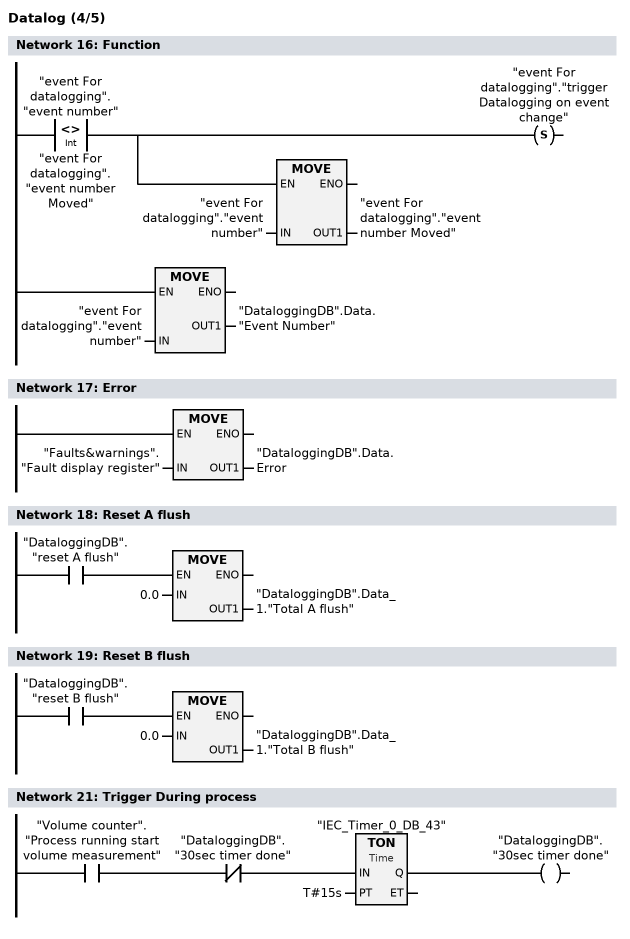
   RUNG wire#powerrail
      { S7_Templates := "SrcType := Int" } NE_Contact(in1 := "event For datalogging"."event number", in2 := "event For datalogging"."event number Moved")
      wire#w1
      S_Coil( "event For datalogging"."trigger Datalogging on event change" )
   END_RUNG
   RUNG wire#w1
      Move(in := "event For datalogging"."event number", out1 => "event For datalogging"."event number Moved")
   END_RUNG
   RUNG wire#powerrail
      Move(in := "event For datalogging"."event number", out1 => "DataloggingDB".Data."Event Number")
   END_RUNG
   // the same network as SCL:
   IF "event For datalogging"."event number" <> "event For datalogging"."event number Moved" THEN
       "event For datalogging"."trigger Datalogging on event change" := TRUE;
       "event For datalogging"."event number Moved" := "event For datalogging"."event number";
   END_IF;
   "DataloggingDB".Data."Event Number" := "event For datalogging"."event number";
END_REGION

REGION Network 17: Error
   RUNG wire#powerrail
      Move(in := "Faults&warnings"."Fault display register", out1 => "DataloggingDB".Data.Error)
   END_RUNG
   // the same network as SCL:
   "DataloggingDB".Data.Error := "Faults&warnings"."Fault display register";
END_REGION

REGION Network 18: Reset A flush
   RUNG wire#powerrail
      Contact( "DataloggingDB"."reset A flush" )
      Move(in := 0.0, out1 => "DataloggingDB".Data_1."Total A flush")
   END_RUNG
   // the same network as SCL:
   IF "DataloggingDB"."reset A flush" THEN "DataloggingDB".Data_1."Total A flush" := 0.0; END_IF;
END_REGION

REGION Network 19: Reset B flush
   RUNG wire#powerrail
      Contact( "DataloggingDB"."reset B flush" )
      Move(in := 0.0, out1 => "DataloggingDB".Data_1."Total B flush")
   END_RUNG
   // the same network as SCL:
   IF "DataloggingDB"."reset B flush" THEN "DataloggingDB".Data_1."Total B flush" := 0.0; END_IF;
END_REGION

REGION Network 20 (SCL): Reset total size
   IF "DataloggingDB"."reset total Size" THEN
       "DataloggingDB".Data_1."Total size A" := 0;
       "DataloggingDB".Data_1."Total size B" := 0;
       "DataloggingDB".totalsizeday := 0;
       "DataloggingDB".totalsizepreviousday := 0;
       "DataloggingDB".totalsizeweek := 0;
       "DataloggingDB".totalsizepreviousweek := 0;
       "DataloggingDB".totalsizemonth := 0;
       "DataloggingDB".totalsizepreviousmonth := 0;
       "DataloggingDB"."reset total Size" := FALSE;
   END_IF;
END_REGION

REGION Network 21: Trigger During process
   RUNG wire#powerrail
      Contact( "Volume counter"."Process running start volume measurement" )
      I_Contact( "DataloggingDB"."30sec timer done" )
      { S7_Templates := "time_type := Time" } "IEC_Timer_0_DB_43".TON(pt := T#15s, et =>)
      Coil( "DataloggingDB"."30sec timer done" )
   END_RUNG
   // the same network as SCL:
   "IEC_Timer_0_DB_43".TON(IN := "Volume counter"."Process running start volume measurement" AND NOT "DataloggingDB"."30sec timer done",
                           PT := T#15s);
   "DataloggingDB"."30sec timer done" := "IEC_Timer_0_DB_43".Q;
END_REGION

REGION Network 22: trigger data logging
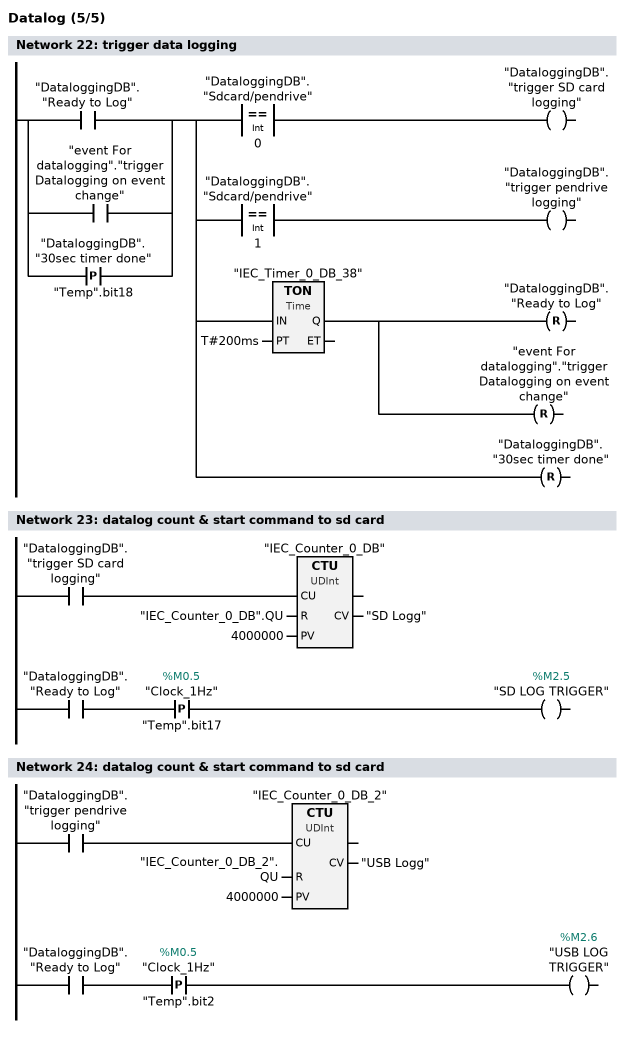
   RUNG wire#powerrail
      Contact( "DataloggingDB"."Ready to Log" )
      wire#w1
      { S7_Templates := "SrcType := Int" } EQ_Contact(in1 := "DataloggingDB"."Sdcard/pendrive", in2 := 0)
      Coil( "DataloggingDB"."trigger SD card logging" )
   END_RUNG
   RUNG wire#powerrail
      Contact( "event For datalogging"."trigger Datalogging on event change" )
   END_RUNG wire#w1
   RUNG wire#powerrail
      P_Contact(operand := "DataloggingDB"."30sec timer done", bit := "Temp".bit18)
   END_RUNG wire#w1
   RUNG wire#w1
      { S7_Templates := "SrcType := Int" } EQ_Contact(in1 := "DataloggingDB"."Sdcard/pendrive", in2 := 1)
      Coil( "DataloggingDB"."trigger pendrive logging" )
   END_RUNG
   RUNG wire#w1
      { S7_Templates := "time_type := Time" } "IEC_Timer_0_DB_38".TON(pt := T#200ms, et =>)
      wire#w2
      R_Coil( "DataloggingDB"."Ready to Log" )
   END_RUNG
   RUNG wire#w2
      R_Coil( "event For datalogging"."trigger Datalogging on event change" )
   END_RUNG
   RUNG wire#w1
      R_Coil( "DataloggingDB"."30sec timer done" )
   END_RUNG
   // the same network as SCL:
   #_w1 := "DataloggingDB"."30sec timer done" AND NOT "Temp".bit18;   // rising edge of "DataloggingDB"."30sec timer done"
   "Temp".bit18 := "DataloggingDB"."30sec timer done";
   #_w2 := "DataloggingDB"."Ready to Log" OR "event For datalogging"."trigger Datalogging on event change" OR #_w1;
   "DataloggingDB"."trigger SD card logging" := #_w2 AND ("DataloggingDB"."Sdcard/pendrive" = 0);
   "DataloggingDB"."trigger pendrive logging" := #_w2 AND ("DataloggingDB"."Sdcard/pendrive" = 1);
   "IEC_Timer_0_DB_38".TON(IN := #_w2, PT := T#200ms);
   IF "IEC_Timer_0_DB_38".Q THEN
       "DataloggingDB"."Ready to Log" := FALSE;
       "event For datalogging"."trigger Datalogging on event change" := FALSE;
   END_IF;
   IF #_w2 THEN "DataloggingDB"."30sec timer done" := FALSE; END_IF;
END_REGION

REGION Network 23: datalog count & start command to sd card
   RUNG wire#powerrail
      Contact( "DataloggingDB"."trigger SD card logging" )
      { S7_Templates := "value_type := UDInt" } "IEC_Counter_0_DB".CTU(r := "IEC_Counter_0_DB".QU, pv := 4000000, cv => "SD Logg")
   END_RUNG
   RUNG wire#powerrail
      Contact( "DataloggingDB"."Ready to Log" )
      P_Contact(operand := "Clock_1Hz", bit := "Temp".bit17)
      Coil( "SD LOG TRIGGER" )
   END_RUNG
   // the same network as SCL:
   "IEC_Counter_0_DB".CTU(CU := "DataloggingDB"."trigger SD card logging",
                          R := "IEC_Counter_0_DB".QU,
                          PV := 4000000,
                          CV => "SD Logg");
   #_w1 := "DataloggingDB"."Ready to Log" AND "Clock_1Hz" AND NOT "Temp".bit17;   // rising edge of "Clock_1Hz"
   "Temp".bit17 := "Clock_1Hz";
   "SD LOG TRIGGER" := #_w1;
END_REGION

REGION Network 24: datalog count & start command to sd card
   RUNG wire#powerrail
      Contact( "DataloggingDB"."trigger pendrive logging" )
      { S7_Templates := "value_type := UDInt" } "IEC_Counter_0_DB_2".CTU(r := "IEC_Counter_0_DB_2".QU, pv := 4000000, cv => "USB Logg")
   END_RUNG
   RUNG wire#powerrail
      Contact( "DataloggingDB"."Ready to Log" )
      P_Contact(operand := "Clock_1Hz", bit := "Temp".bit2)
      Coil( "USB LOG TRIGGER" )
   END_RUNG
   // the same network as SCL:
   "IEC_Counter_0_DB_2".CTU(CU := "DataloggingDB"."trigger pendrive logging",
                           R := "IEC_Counter_0_DB_2".QU,
                           PV := 4000000,
                           CV => "USB Logg");
   #_w1 := "DataloggingDB"."Ready to Log" AND "Clock_1Hz" AND NOT "Temp".bit2;   // rising edge of "Clock_1Hz"
   "Temp".bit2 := "Clock_1Hz";
   "USB LOG TRIGGER" := #_w1;
END_REGION
END_FUNCTION

FUNCTION "IOT_DATA_FC" : Void   // FC1001, LAD
{ S7_Optimized_Access := 'TRUE' }
VERSION : 0.1
// stored: AutoNumber false, IsIECCheckEnabled true, SetENOAutomatically true, UDAEnableTagReadback false
BEGIN

REGION Network 1 (SCL)
   "IOT_DATA"."pump A Inlet" := "pressure"."pump A Inlet";
   "IOT_DATA"."pump B Inlet" := "pressure"."pump B Inlet";
   "IOT_DATA"."pump A Outlet" := "pressure"."pump A Outlet";
   "IOT_DATA"."pump B Outlet" := "pressure"."pump B Outlet";
END_REGION
END_FUNCTION

FUNCTION "Output_Estop" : Void   // FC31, LAD
{ S7_Optimized_Access := 'TRUE' }
VERSION : 0.1
// stored: AutoNumber true, IsIECCheckEnabled false, SetENOAutomatically false, UDAEnableTagReadback false
   VAR_TEMP
      spare : Bool;
      spare2 : Bool;
      spare3 : Bool;
   END_VAR
BEGIN

REGION Network 1: gear Pump A
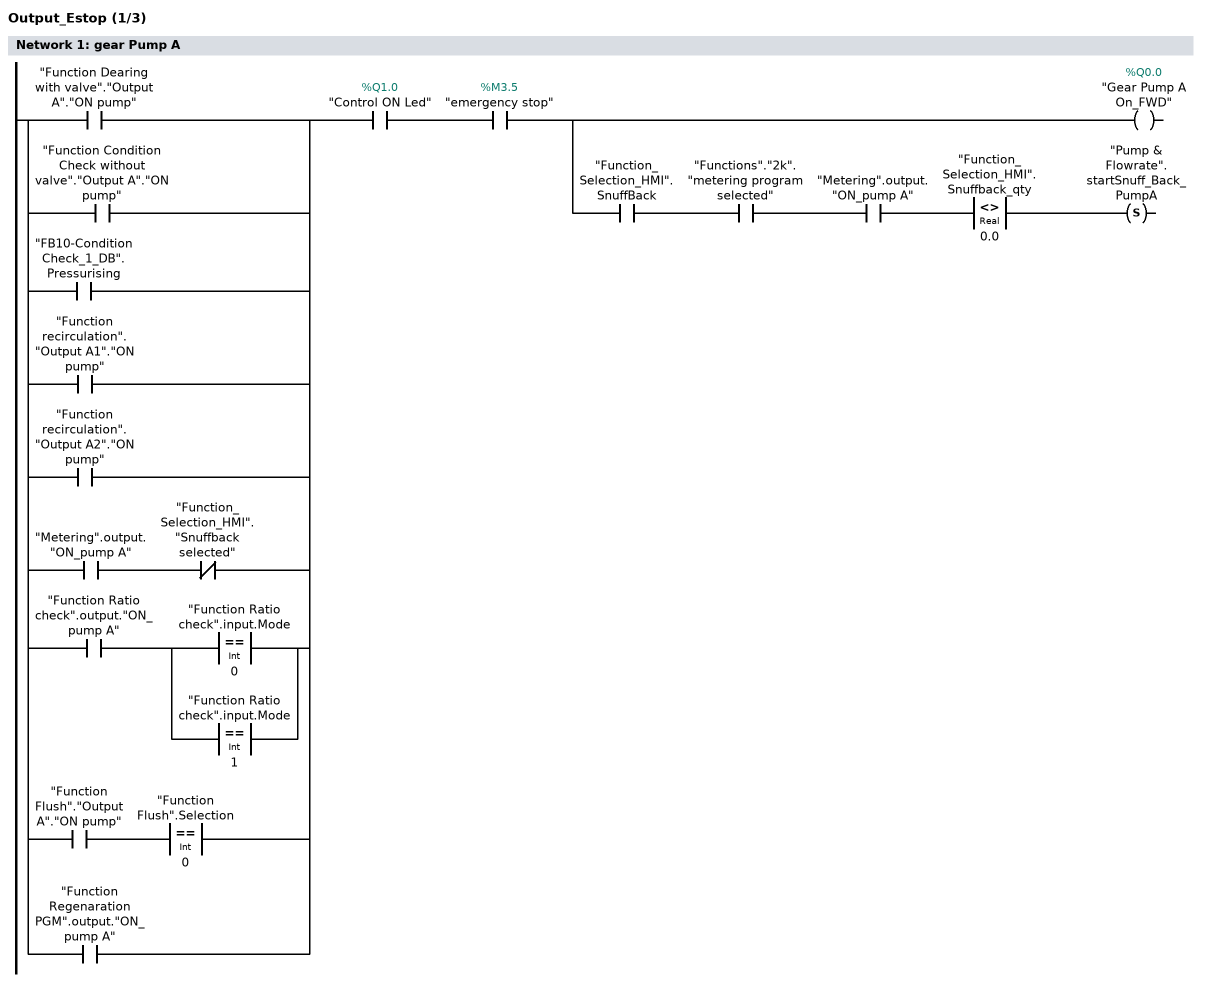
   RUNG wire#powerrail
      Contact( "Function Dearing with valve"."Output A"."ON pump" )
      wire#w1
      Contact( "Control ON Led" )
      Contact( "emergency stop" )
      wire#w3
      Coil( "Gear Pump A On_FWD" )
   END_RUNG
   RUNG wire#powerrail
      Contact( "Function ConditionCheck without valve"."Output A"."ON pump" )
   END_RUNG wire#w1
   RUNG wire#powerrail
      Contact( "FB10-Condition Check_1_DB".Pressurising )
   END_RUNG wire#w1
   RUNG wire#powerrail
      Contact( "Function recirculation"."Output A1"."ON pump" )
   END_RUNG wire#w1
   RUNG wire#powerrail
      Contact( "Function recirculation"."Output A2"."ON pump" )
   END_RUNG wire#w1
   RUNG wire#powerrail
      Contact( "Metering".output."ON_pump A" )
      I_Contact( "Function_Selection_HMI"."Snuffback selected" )
   END_RUNG wire#w1
   RUNG wire#powerrail
      Contact( "Function Ratio check".output."ON_pump A" )
      wire#w2
      { S7_Templates := "SrcType := Int" } EQ_Contact(in1 := "Function Ratio check".input.Mode, in2 := 0)
   END_RUNG wire#w1
   RUNG wire#w2
      { S7_Templates := "SrcType := Int" } EQ_Contact(in1 := "Function Ratio check".input.Mode, in2 := 1)
   END_RUNG wire#w1
   RUNG wire#powerrail
      Contact( "Function Flush"."Output A"."ON pump" )
      { S7_Templates := "SrcType := Int" } EQ_Contact(in1 := "Function Flush".Selection, in2 := 0)
   END_RUNG wire#w1
   RUNG wire#powerrail
      Contact( "Function Regenaration PGM".output."ON_pump A" )
   END_RUNG wire#w1
   RUNG wire#w3
      Contact( "Function_Selection_HMI".SnuffBack )
      Contact( "Functions"."2k"."metering program selected" )
      Contact( "Metering".output."ON_pump A" )
      { S7_Templates := "SrcType := Real" } NE_Contact(in1 := "Function_Selection_HMI".Snuffback_qty, in2 := 0.0)
      S_Coil( "Pump & Flowrate".startSnuff_Back_PumpA )
   END_RUNG
   // the same network as SCL:
   "Gear Pump A On_FWD" := ("Function Dearing with valve"."Output A"."ON pump" OR "Function ConditionCheck without valve"."Output A"."ON pump" OR "FB10-Condition Check_1_DB".Pressurising OR "Function recirculation"."Output A1"."ON pump" OR "Function recirculation"."Output A2"."ON pump" OR ("Metering".output."ON_pump A" AND NOT "Function_Selection_HMI"."Snuffback selected") OR ("Function Ratio check".output."ON_pump A" AND (("Function Ratio check".input.Mode = 0) OR ("Function Ratio check".input.Mode = 1))) OR ("Function Flush"."Output A"."ON pump" AND ("Function Flush".Selection = 0)) OR "Function Regenaration PGM".output."ON_pump A") AND "Control ON Led" AND "emergency stop";
   IF "Gear Pump A On_FWD" AND "Function_Selection_HMI".SnuffBack AND "Functions"."2k"."metering program selected" AND "Metering".output."ON_pump A" AND ("Function_Selection_HMI".Snuffback_qty <> 0.0) THEN
       "Pump & Flowrate".startSnuff_Back_PumpA := TRUE;
   END_IF;
END_REGION

REGION Network 2: gear Pump B
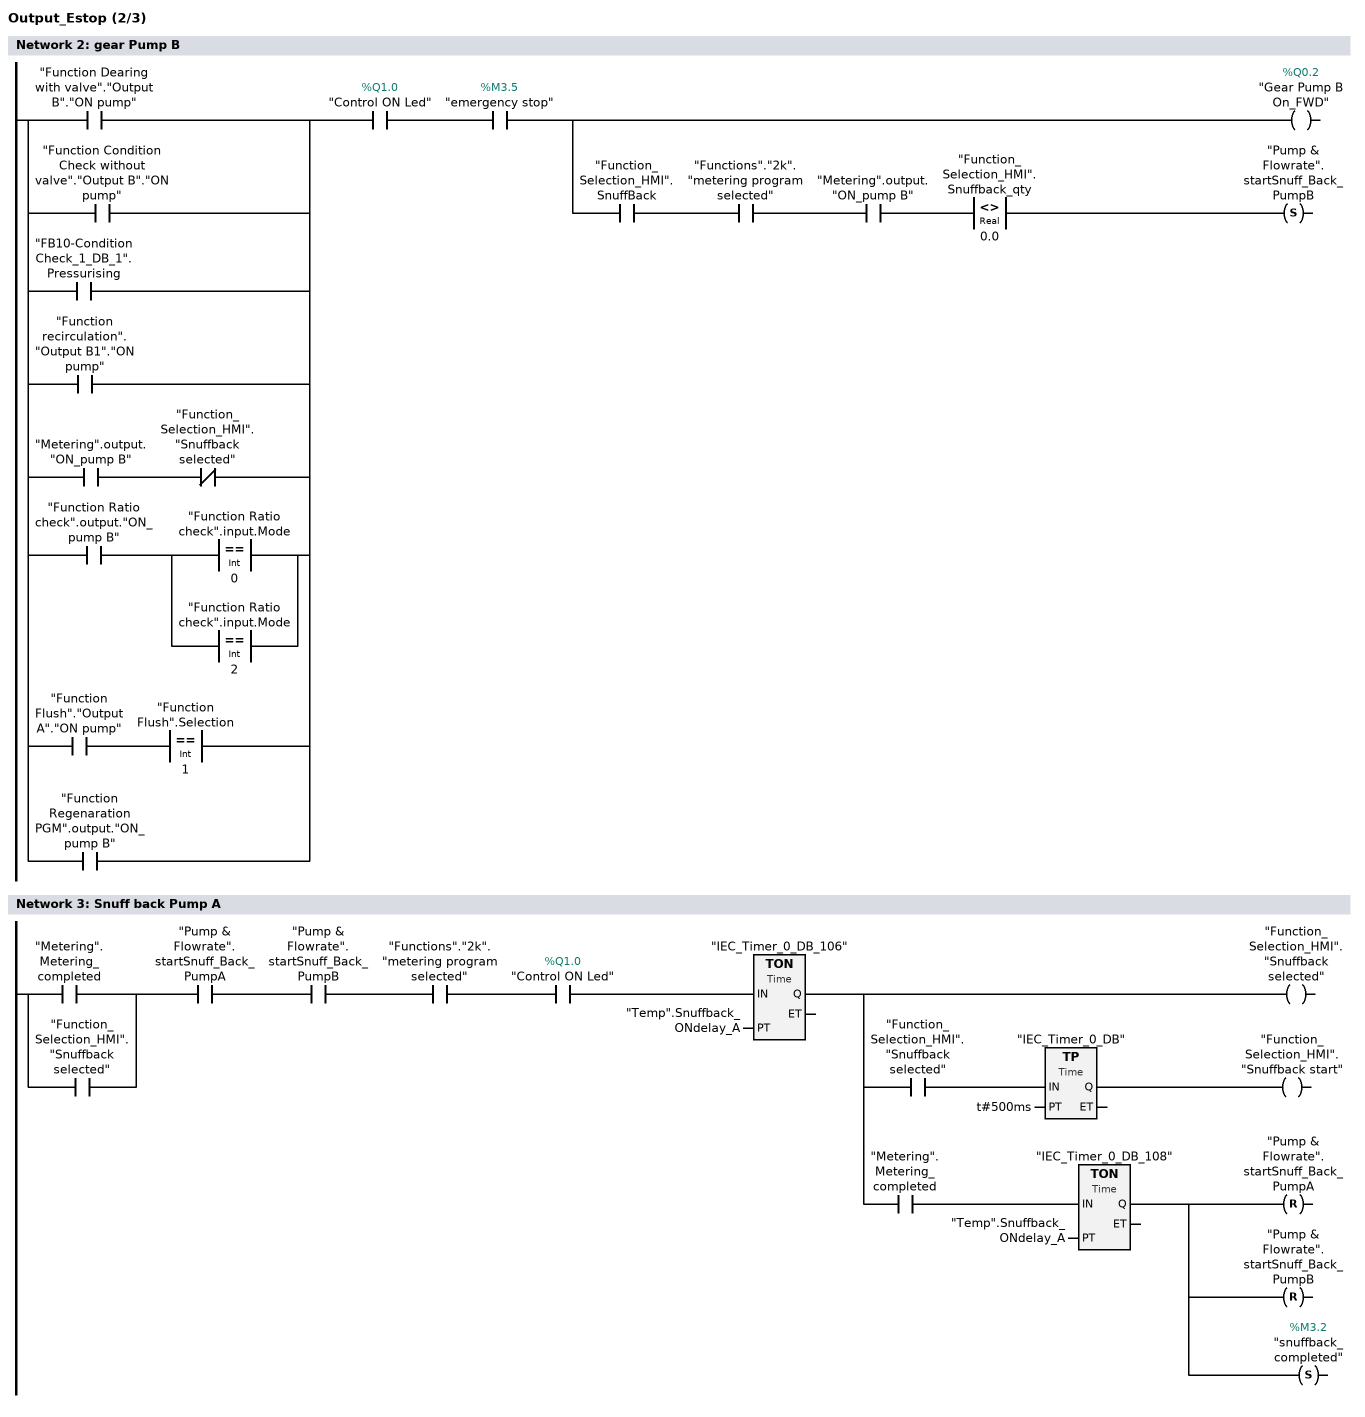
   RUNG wire#powerrail
      Contact( "Function Dearing with valve"."Output B"."ON pump" )
      wire#w1
      Contact( "Control ON Led" )
      Contact( "emergency stop" )
      wire#w3
      Coil( "Gear Pump B On_FWD" )
   END_RUNG
   RUNG wire#powerrail
      Contact( "Function ConditionCheck without valve"."Output B"."ON pump" )
   END_RUNG wire#w1
   RUNG wire#powerrail
      Contact( "FB10-Condition Check_1_DB_1".Pressurising )
   END_RUNG wire#w1
   RUNG wire#powerrail
      Contact( "Function recirculation"."Output B1"."ON pump" )
   END_RUNG wire#w1
   RUNG wire#powerrail
      Contact( "Metering".output."ON_pump B" )
      I_Contact( "Function_Selection_HMI"."Snuffback selected" )
   END_RUNG wire#w1
   RUNG wire#powerrail
      Contact( "Function Ratio check".output."ON_pump B" )
      wire#w2
      { S7_Templates := "SrcType := Int" } EQ_Contact(in1 := "Function Ratio check".input.Mode, in2 := 0)
   END_RUNG wire#w1
   RUNG wire#w2
      { S7_Templates := "SrcType := Int" } EQ_Contact(in1 := "Function Ratio check".input.Mode, in2 := 2)
   END_RUNG wire#w1
   RUNG wire#powerrail
      Contact( "Function Flush"."Output A"."ON pump" )
      { S7_Templates := "SrcType := Int" } EQ_Contact(in1 := "Function Flush".Selection, in2 := 1)
   END_RUNG wire#w1
   RUNG wire#powerrail
      Contact( "Function Regenaration PGM".output."ON_pump B" )
   END_RUNG wire#w1
   RUNG wire#w3
      Contact( "Function_Selection_HMI".SnuffBack )
      Contact( "Functions"."2k"."metering program selected" )
      Contact( "Metering".output."ON_pump B" )
      { S7_Templates := "SrcType := Real" } NE_Contact(in1 := "Function_Selection_HMI".Snuffback_qty, in2 := 0.0)
      S_Coil( "Pump & Flowrate".startSnuff_Back_PumpB )
   END_RUNG
   // the same network as SCL:
   "Gear Pump B On_FWD" := ("Function Dearing with valve"."Output B"."ON pump" OR "Function ConditionCheck without valve"."Output B"."ON pump" OR "FB10-Condition Check_1_DB_1".Pressurising OR "Function recirculation"."Output B1"."ON pump" OR ("Metering".output."ON_pump B" AND NOT "Function_Selection_HMI"."Snuffback selected") OR ("Function Ratio check".output."ON_pump B" AND (("Function Ratio check".input.Mode = 0) OR ("Function Ratio check".input.Mode = 2))) OR ("Function Flush"."Output A"."ON pump" AND ("Function Flush".Selection = 1)) OR "Function Regenaration PGM".output."ON_pump B") AND "Control ON Led" AND "emergency stop";
   IF "Gear Pump B On_FWD" AND "Function_Selection_HMI".SnuffBack AND "Functions"."2k"."metering program selected" AND "Metering".output."ON_pump B" AND ("Function_Selection_HMI".Snuffback_qty <> 0.0) THEN
       "Pump & Flowrate".startSnuff_Back_PumpB := TRUE;
   END_IF;
END_REGION

REGION Network 3: Snuff back Pump A
   RUNG wire#powerrail
      Contact( "Metering".Metering_completed )
      wire#w1
      Contact( "Pump & Flowrate".startSnuff_Back_PumpA )
      Contact( "Pump & Flowrate".startSnuff_Back_PumpB )
      Contact( "Functions"."2k"."metering program selected" )
      Contact( "Control ON Led" )
      { S7_Templates := "time_type := Time" } "IEC_Timer_0_DB_106".TON(pt := "Temp".Snuffback_ONdelay_A, et =>)
      wire#w2
      Coil( "Function_Selection_HMI"."Snuffback selected" )
   END_RUNG
   RUNG wire#powerrail
      Contact( "Function_Selection_HMI"."Snuffback selected" )
   END_RUNG wire#w1
   RUNG wire#w2
      Contact( "Function_Selection_HMI"."Snuffback selected" )
      { S7_Templates := "time_type := Time" } "IEC_Timer_0_DB".TP(pt := t#500ms, et =>)
      Coil( "Function_Selection_HMI"."Snuffback start" )
   END_RUNG
   RUNG wire#w2
      Contact( "Metering".Metering_completed )
      { S7_Templates := "time_type := Time" } "IEC_Timer_0_DB_108".TON(pt := "Temp".Snuffback_ONdelay_A, et =>)
      wire#w3
      R_Coil( "Pump & Flowrate".startSnuff_Back_PumpA )
   END_RUNG
   RUNG wire#w3
      R_Coil( "Pump & Flowrate".startSnuff_Back_PumpB )
   END_RUNG
   RUNG wire#w3
      S_Coil( "snuffback_completed" )
   END_RUNG
   // the same network as SCL:
   "IEC_Timer_0_DB_106".TON(IN := ("Metering".Metering_completed OR "Function_Selection_HMI"."Snuffback selected") AND "Pump & Flowrate".startSnuff_Back_PumpA AND "Pump & Flowrate".startSnuff_Back_PumpB AND "Functions"."2k"."metering program selected" AND "Control ON Led",
                           PT := "Temp".Snuffback_ONdelay_A);
   "Function_Selection_HMI"."Snuffback selected" := "IEC_Timer_0_DB_106".Q;
   "IEC_Timer_0_DB".TP(IN := "IEC_Timer_0_DB_106".Q AND "Function_Selection_HMI"."Snuffback selected",
                       PT := t#500ms);
   "Function_Selection_HMI"."Snuffback start" := "IEC_Timer_0_DB".Q;
   "IEC_Timer_0_DB_108".TON(IN := "IEC_Timer_0_DB_106".Q AND "Metering".Metering_completed,
                           PT := "Temp".Snuffback_ONdelay_A);
   IF "IEC_Timer_0_DB_108".Q THEN
       "Pump & Flowrate".startSnuff_Back_PumpA := FALSE;
       "Pump & Flowrate".startSnuff_Back_PumpB := FALSE;
       "snuffback_completed" := TRUE;
   END_IF;
END_REGION

REGION Network 4
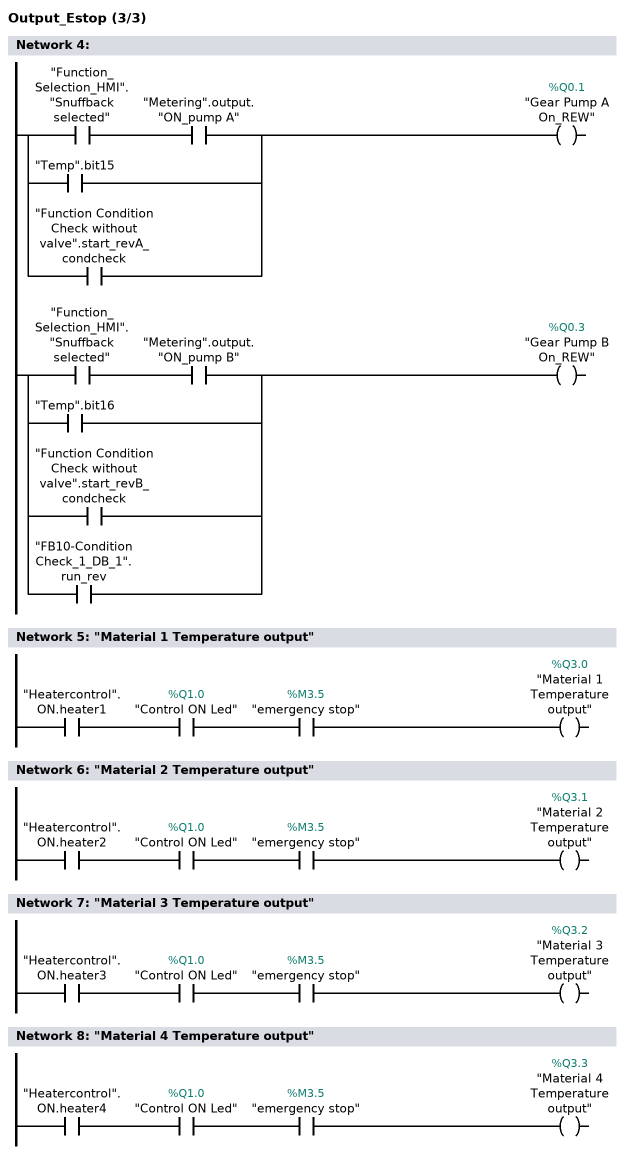
   RUNG wire#powerrail
      Contact( "Function_Selection_HMI"."Snuffback selected" )
      Contact( "Metering".output."ON_pump A" )
      wire#w1
      Coil( "Gear Pump A On_REW" )
   END_RUNG
   RUNG wire#powerrail
      Contact( "Temp".bit15 )
   END_RUNG wire#w1
   RUNG wire#powerrail
      Contact( "Function ConditionCheck without valve".start_revA_condcheck )
   END_RUNG wire#w1
   RUNG wire#powerrail
      Contact( "Function_Selection_HMI"."Snuffback selected" )
      Contact( "Metering".output."ON_pump B" )
      wire#w2
      Coil( "Gear Pump B On_REW" )
   END_RUNG
   RUNG wire#powerrail
      Contact( "Temp".bit16 )
   END_RUNG wire#w2
   RUNG wire#powerrail
      Contact( "Function ConditionCheck without valve".start_revB_condcheck )
   END_RUNG wire#w2
   RUNG wire#powerrail
      Contact( "FB10-Condition Check_1_DB_1".run_rev )
   END_RUNG wire#w2
   // the same network as SCL:
   "Gear Pump A On_REW" := ("Function_Selection_HMI"."Snuffback selected" AND "Metering".output."ON_pump A") OR "Temp".bit15 OR "Function ConditionCheck without valve".start_revA_condcheck;
   "Gear Pump B On_REW" := ("Function_Selection_HMI"."Snuffback selected" AND "Metering".output."ON_pump B") OR "Temp".bit16 OR "Function ConditionCheck without valve".start_revB_condcheck OR "FB10-Condition Check_1_DB_1".run_rev;
END_REGION

REGION Network 5: "Material 1 Temperature output"
   RUNG wire#powerrail
      Contact( "Heatercontrol".ON.heater1 )
      Contact( "Control ON Led" )
      Contact( "emergency stop" )
      Coil( "Material 1 Temperature output" )
   END_RUNG
   // the same network as SCL:
   "Material 1 Temperature output" := "Heatercontrol".ON.heater1 AND "Control ON Led" AND "emergency stop";
END_REGION

REGION Network 6: "Material 2 Temperature output"
   RUNG wire#powerrail
      Contact( "Heatercontrol".ON.heater2 )
      Contact( "Control ON Led" )
      Contact( "emergency stop" )
      Coil( "Material 2 Temperature output" )
   END_RUNG
   // the same network as SCL:
   "Material 2 Temperature output" := "Heatercontrol".ON.heater2 AND "Control ON Led" AND "emergency stop";
END_REGION

REGION Network 7: "Material 3 Temperature output"
   RUNG wire#powerrail
      Contact( "Heatercontrol".ON.heater3 )
      Contact( "Control ON Led" )
      Contact( "emergency stop" )
      Coil( "Material 3 Temperature output" )
   END_RUNG
   // the same network as SCL:
   "Material 3 Temperature output" := "Heatercontrol".ON.heater3 AND "Control ON Led" AND "emergency stop";
END_REGION

REGION Network 8: "Material 4 Temperature output"
   RUNG wire#powerrail
      Contact( "Heatercontrol".ON.heater4 )
      Contact( "Control ON Led" )
      Contact( "emergency stop" )
      Coil( "Material 4 Temperature output" )
   END_RUNG
   // the same network as SCL:
   "Material 4 Temperature output" := "Heatercontrol".ON.heater4 AND "Control ON Led" AND "emergency stop";
END_REGION
END_FUNCTION

FUNCTION "Conditon Check" : Void   // FC11, LAD
{ S7_Optimized_Access := 'TRUE' }
VERSION : 0.1
// stored: AutoNumber true, IsIECCheckEnabled false, SetENOAutomatically false, UDAEnableTagReadback false
   VAR_TEMP   // added for the SCL form of the ladder/FBD networks
      _w1 : Bool;
      _w2 : Bool;
      _w3 : Bool;
   END_VAR
BEGIN

REGION Network 1: Condition Check A without Valve
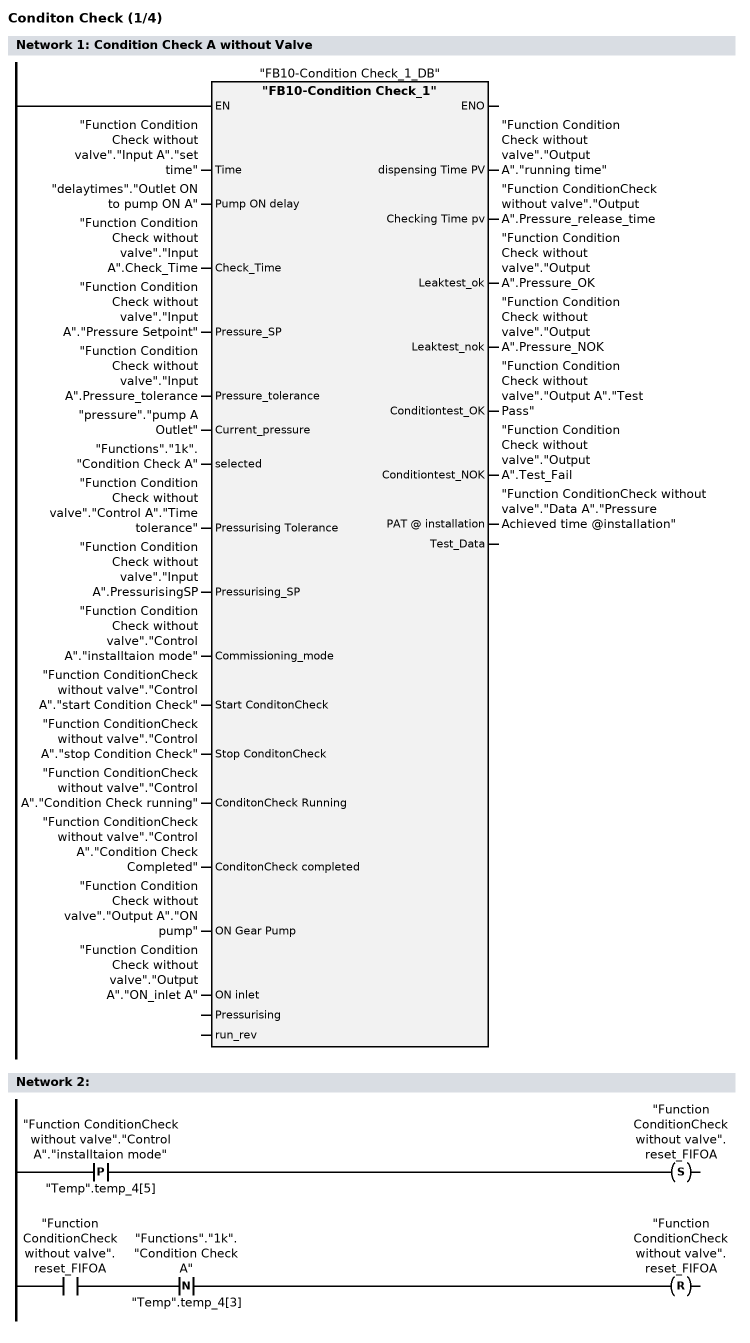
   RUNG wire#powerrail
      "FB10-Condition Check_1_DB"("Time" := "Function ConditionCheck without valve"."Input A"."set time", "Pump ON delay" := "delaytimes"."Outlet ON to pump ON A", Check_Time := "Function ConditionCheck without valve"."Input A".Check_Time, Pressure_SP := "Function ConditionCheck without valve"."Input A"."Pressure Setpoint", Pressure_tolerance := "Function ConditionCheck without valve"."Input A".Pressure_tolerance, Current_pressure := "pressure"."pump A Outlet", selected := "Functions"."1k"."Condition Check A", "Pressurising Tolerance" := "Function ConditionCheck without valve"."Control A"."Time tolerance", Pressurising_SP := "Function ConditionCheck without valve"."Input A".PressurisingSP, Commissioning_mode := "Function ConditionCheck without valve"."Control A"."installtaion mode", "Start ConditonCheck" := "Function ConditionCheck without valve"."Control A"."start Condition Check", "Stop ConditonCheck" := "Function ConditionCheck without valve"."Control A"."stop Condition Check", "ConditonCheck Running" := "Function ConditionCheck without valve"."Control A"."Condition Check running", "ConditonCheck completed" := "Function ConditionCheck without valve"."Control A"."Condition Check Completed", "ON Gear Pump" := "Function ConditionCheck without valve"."Output A"."ON pump", "ON inlet" := "Function ConditionCheck without valve"."Output A"."ON_inlet A", Pressurising :=, run_rev :=, "dispensing Time PV" => "Function ConditionCheck without valve"."Output A"."running time", "Checking Time pv" => "Function ConditionCheck without valve"."Output A".Pressure_release_time, Leaktest_ok => "Function ConditionCheck without valve"."Output A".Pressure_OK, Leaktest_nok => "Function ConditionCheck without valve"."Output A".Pressure_NOK, Conditiontest_OK => "Function ConditionCheck without valve"."Output A"."Test Pass", Conditiontest_NOK => "Function ConditionCheck without valve"."Output A".Test_Fail, "PAT @ installation" => "Function ConditionCheck without valve"."Data A"."Pressure Achieved time @installation", Test_Data =>)
   END_RUNG
   // the same network as SCL:
   "FB10-Condition Check_1_DB"("Time" := "Function ConditionCheck without valve"."Input A"."set time",   // "FB10-Condition Check_1"
                           "Pump ON delay" := "delaytimes"."Outlet ON to pump ON A",
                           Check_Time := "Function ConditionCheck without valve"."Input A".Check_Time,
                           Pressure_SP := "Function ConditionCheck without valve"."Input A"."Pressure Setpoint",
                           Pressure_tolerance := "Function ConditionCheck without valve"."Input A".Pressure_tolerance,
                           Current_pressure := "pressure"."pump A Outlet",
                           selected := "Functions"."1k"."Condition Check A",
                           "Pressurising Tolerance" := "Function ConditionCheck without valve"."Control A"."Time tolerance",
                           Pressurising_SP := "Function ConditionCheck without valve"."Input A".PressurisingSP,
                           Commissioning_mode := "Function ConditionCheck without valve"."Control A"."installtaion mode",
                           "Start ConditonCheck" := "Function ConditionCheck without valve"."Control A"."start Condition Check",
                           "Stop ConditonCheck" := "Function ConditionCheck without valve"."Control A"."stop Condition Check",
                           "ConditonCheck Running" := "Function ConditionCheck without valve"."Control A"."Condition Check running",
                           "ConditonCheck completed" := "Function ConditionCheck without valve"."Control A"."Condition Check Completed",
                           "ON Gear Pump" := "Function ConditionCheck without valve"."Output A"."ON pump",
                           "ON inlet" := "Function ConditionCheck without valve"."Output A"."ON_inlet A",
                           "dispensing Time PV" => "Function ConditionCheck without valve"."Output A"."running time",
                           "Checking Time pv" => "Function ConditionCheck without valve"."Output A".Pressure_release_time,
                           Leaktest_ok => "Function ConditionCheck without valve"."Output A".Pressure_OK,
                           Leaktest_nok => "Function ConditionCheck without valve"."Output A".Pressure_NOK,
                           Conditiontest_OK => "Function ConditionCheck without valve"."Output A"."Test Pass",
                           Conditiontest_NOK => "Function ConditionCheck without valve"."Output A".Test_Fail,
                           "PAT @ installation" => "Function ConditionCheck without valve"."Data A"."Pressure Achieved time @installation");
END_REGION

REGION Network 2
   RUNG wire#powerrail
      P_Contact(operand := "Function ConditionCheck without valve"."Control A"."installtaion mode", bit := "Temp".temp_4[5])
      S_Coil( "Function ConditionCheck without valve".reset_FIFOA )
   END_RUNG
   RUNG wire#powerrail
      Contact( "Function ConditionCheck without valve".reset_FIFOA )
      N_Contact(operand := "Functions"."1k"."Condition Check A", bit := "Temp".temp_4[3])
      R_Coil( "Function ConditionCheck without valve".reset_FIFOA )
   END_RUNG
   // the same network as SCL:
   #_w1 := "Function ConditionCheck without valve"."Control A"."installtaion mode" AND NOT "Temp".temp_4[5];   // rising edge of "Function ConditionCheck without valve"."Control A"."installtaion mode"
   "Temp".temp_4[5] := "Function ConditionCheck without valve"."Control A"."installtaion mode";
   IF #_w1 THEN "Function ConditionCheck without valve".reset_FIFOA := TRUE; END_IF;
   #_w2 := "Function ConditionCheck without valve".reset_FIFOA AND NOT "Functions"."1k"."Condition Check A" AND "Temp".temp_4[3];   // falling edge of "Functions"."1k"."Condition Check A"
   "Temp".temp_4[3] := "Functions"."1k"."Condition Check A";
   IF #_w2 THEN "Function ConditionCheck without valve".reset_FIFOA := FALSE; END_IF;
END_REGION

REGION Network 3
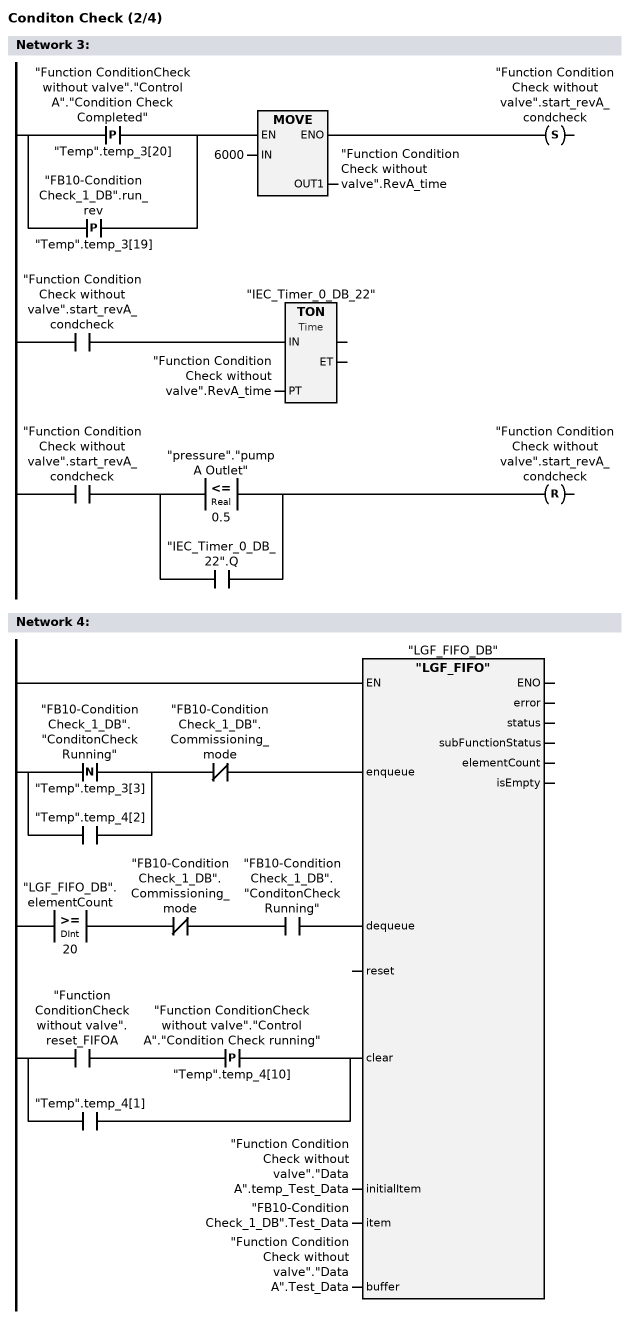
   RUNG wire#powerrail
      P_Contact(operand := "Function ConditionCheck without valve"."Control A"."Condition Check Completed", bit := "Temp".temp_3[20])
      wire#w1
      Move(in := 6000, out1 => "Function ConditionCheck without valve".RevA_time)
      S_Coil( "Function ConditionCheck without valve".start_revA_condcheck )
   END_RUNG
   RUNG wire#powerrail
      P_Contact(operand := "FB10-Condition Check_1_DB".run_rev, bit := "Temp".temp_3[19])
   END_RUNG wire#w1
   RUNG wire#powerrail
      Contact( "Function ConditionCheck without valve".start_revA_condcheck )
      { S7_Templates := "time_type := Time" } "IEC_Timer_0_DB_22".TON(pt := "Function ConditionCheck without valve".RevA_time, et =>)
   END_RUNG
   RUNG wire#powerrail
      Contact( "Function ConditionCheck without valve".start_revA_condcheck )
      wire#w2
      { S7_Templates := "SrcType := Real" } LE_Contact(in1 := "pressure"."pump A Outlet", in2 := 0.5)
      wire#w3
      R_Coil( "Function ConditionCheck without valve".start_revA_condcheck )
   END_RUNG
   RUNG wire#w2
      Contact( "IEC_Timer_0_DB_22".Q )
   END_RUNG wire#w3
   // the same network as SCL:
   #_w1 := "Function ConditionCheck without valve"."Control A"."Condition Check Completed" AND NOT "Temp".temp_3[20];   // rising edge of "Function ConditionCheck without valve"."Control A"."Condition Check Completed"
   "Temp".temp_3[20] := "Function ConditionCheck without valve"."Control A"."Condition Check Completed";
   #_w2 := "FB10-Condition Check_1_DB".run_rev AND NOT "Temp".temp_3[19];   // rising edge of "FB10-Condition Check_1_DB".run_rev
   "Temp".temp_3[19] := "FB10-Condition Check_1_DB".run_rev;
   IF #_w1 OR #_w2 THEN
       "Function ConditionCheck without valve".RevA_time := 6000;
       "Function ConditionCheck without valve".start_revA_condcheck := TRUE;
   END_IF;
   "IEC_Timer_0_DB_22".TON(IN := "Function ConditionCheck without valve".start_revA_condcheck,
                           PT := "Function ConditionCheck without valve".RevA_time);
   IF "Function ConditionCheck without valve".start_revA_condcheck AND (("pressure"."pump A Outlet" <= 0.5) OR "IEC_Timer_0_DB_22".Q) THEN
       "Function ConditionCheck without valve".start_revA_condcheck := FALSE;
   END_IF;
END_REGION

REGION Network 4
   RUNG wire#powerrail
      "LGF_FIFO_DB"(enqueue := wire#w2, dequeue := wire#w3, clear := wire#w4, reset :=, initialItem := "Function ConditionCheck without valve"."Data A".temp_Test_Data, item := "FB10-Condition Check_1_DB".Test_Data, buffer := "Function ConditionCheck without valve"."Data A".Test_Data, error =>, status =>, subFunctionStatus =>, elementCount =>, isEmpty =>)
   END_RUNG
   RUNG wire#powerrail
      N_Contact(operand := "FB10-Condition Check_1_DB"."ConditonCheck Running", bit := "Temp".temp_3[3])
      wire#w1
      I_Contact( "FB10-Condition Check_1_DB".Commissioning_mode )
   END_RUNG wire#w2
   RUNG wire#powerrail
      Contact( "Temp".temp_4[2] )
   END_RUNG wire#w1
   RUNG wire#powerrail
      { S7_Templates := "SrcType := DInt" } GE_Contact(in1 := "LGF_FIFO_DB".elementCount, in2 := 20)
      I_Contact( "FB10-Condition Check_1_DB".Commissioning_mode )
      Contact( "FB10-Condition Check_1_DB"."ConditonCheck Running" )
   END_RUNG wire#w3
   RUNG wire#powerrail
      Contact( "Function ConditionCheck without valve".reset_FIFOA )
      P_Contact(operand := "Function ConditionCheck without valve"."Control A"."Condition Check running", bit := "Temp".temp_4[10])
   END_RUNG wire#w4
   RUNG wire#powerrail
      Contact( "Temp".temp_4[1] )
   END_RUNG wire#w4
   // the same network as SCL:
   #_w1 := NOT "FB10-Condition Check_1_DB"."ConditonCheck Running" AND "Temp".temp_3[3];   // falling edge of "FB10-Condition Check_1_DB"."ConditonCheck Running"
   "Temp".temp_3[3] := "FB10-Condition Check_1_DB"."ConditonCheck Running";
   #_w3 := (#_w1 OR "Temp".temp_4[2]) AND NOT "FB10-Condition Check_1_DB".Commissioning_mode;
   #_w2 := "Function ConditionCheck without valve".reset_FIFOA AND "Function ConditionCheck without valve"."Control A"."Condition Check running" AND NOT "Temp".temp_4[10];   // rising edge of "Function ConditionCheck without valve"."Control A"."Condition Check running"
   "Temp".temp_4[10] := "Function ConditionCheck without valve"."Control A"."Condition Check running";
   "LGF_FIFO_DB"(enqueue := #_w3,   // "LGF_FIFO"
                 dequeue := ("LGF_FIFO_DB".elementCount >= 20) AND NOT "FB10-Condition Check_1_DB".Commissioning_mode AND "FB10-Condition Check_1_DB"."ConditonCheck Running",
                 clear := #_w2 OR "Temp".temp_4[1],
                 initialItem := "Function ConditionCheck without valve"."Data A".temp_Test_Data,
                 item := "FB10-Condition Check_1_DB".Test_Data,
                 buffer := "Function ConditionCheck without valve"."Data A".Test_Data);
END_REGION

REGION Network 5: Condition Check B without Valve
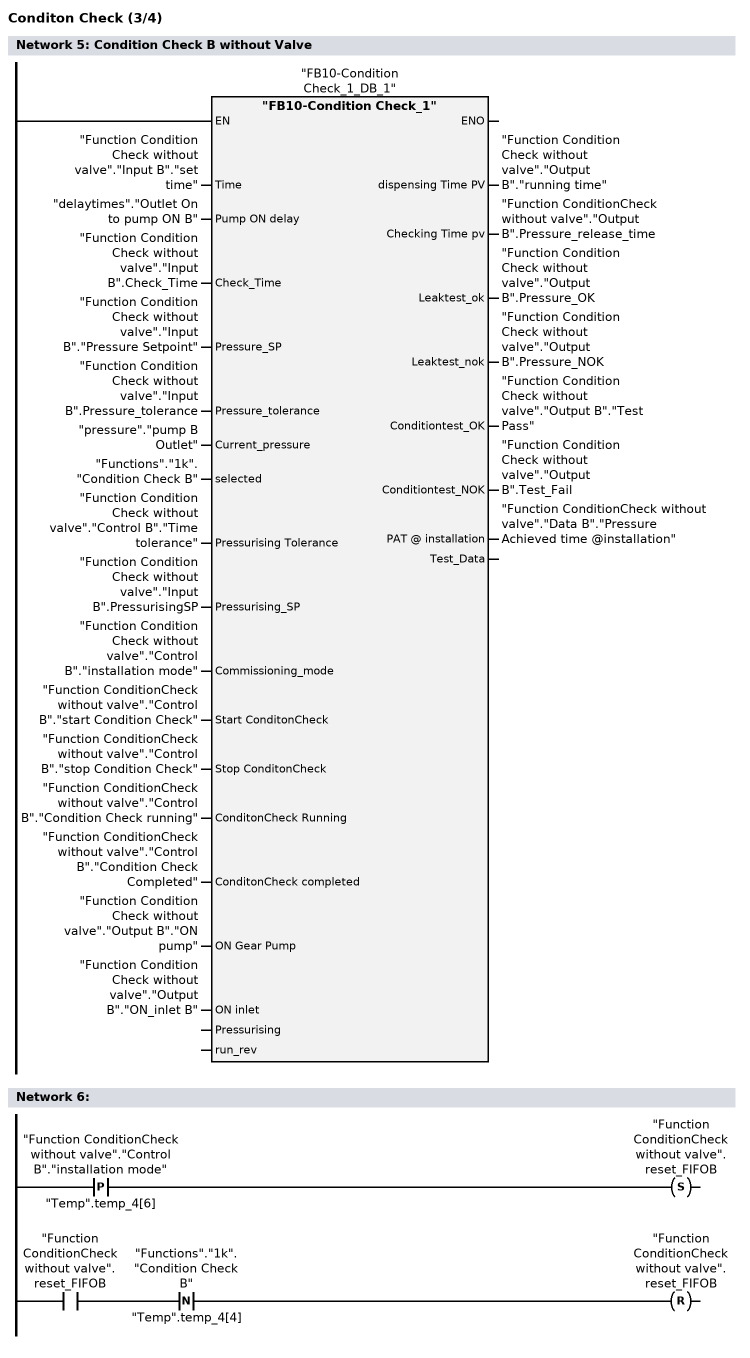
   RUNG wire#powerrail
      "FB10-Condition Check_1_DB_1"("Time" := "Function ConditionCheck without valve"."Input B"."set time", "Pump ON delay" := "delaytimes"."Outlet On to pump ON B", Check_Time := "Function ConditionCheck without valve"."Input B".Check_Time, Pressure_SP := "Function ConditionCheck without valve"."Input B"."Pressure Setpoint", Pressure_tolerance := "Function ConditionCheck without valve"."Input B".Pressure_tolerance, Current_pressure := "pressure"."pump B Outlet", selected := "Functions"."1k"."Condition Check B", "Pressurising Tolerance" := "Function ConditionCheck without valve"."Control B"."Time tolerance", Pressurising_SP := "Function ConditionCheck without valve"."Input B".PressurisingSP, Commissioning_mode := "Function ConditionCheck without valve"."Control B"."installation mode", "Start ConditonCheck" := "Function ConditionCheck without valve"."Control B"."start Condition Check", "Stop ConditonCheck" := "Function ConditionCheck without valve"."Control B"."stop Condition Check", "ConditonCheck Running" := "Function ConditionCheck without valve"."Control B"."Condition Check running", "ConditonCheck completed" := "Function ConditionCheck without valve"."Control B"."Condition Check Completed", "ON Gear Pump" := "Function ConditionCheck without valve"."Output B"."ON pump", "ON inlet" := "Function ConditionCheck without valve"."Output B"."ON_inlet B", Pressurising :=, run_rev :=, "dispensing Time PV" => "Function ConditionCheck without valve"."Output B"."running time", "Checking Time pv" => "Function ConditionCheck without valve"."Output B".Pressure_release_time, Leaktest_ok => "Function ConditionCheck without valve"."Output B".Pressure_OK, Leaktest_nok => "Function ConditionCheck without valve"."Output B".Pressure_NOK, Conditiontest_OK => "Function ConditionCheck without valve"."Output B"."Test Pass", Conditiontest_NOK => "Function ConditionCheck without valve"."Output B".Test_Fail, "PAT @ installation" => "Function ConditionCheck without valve"."Data B"."Pressure Achieved time @installation", Test_Data =>)
   END_RUNG
   // the same network as SCL:
   "FB10-Condition Check_1_DB_1"("Time" := "Function ConditionCheck without valve"."Input B"."set time",   // "FB10-Condition Check_1"
                           "Pump ON delay" := "delaytimes"."Outlet On to pump ON B",
                           Check_Time := "Function ConditionCheck without valve"."Input B".Check_Time,
                           Pressure_SP := "Function ConditionCheck without valve"."Input B"."Pressure Setpoint",
                           Pressure_tolerance := "Function ConditionCheck without valve"."Input B".Pressure_tolerance,
                           Current_pressure := "pressure"."pump B Outlet",
                           selected := "Functions"."1k"."Condition Check B",
                           "Pressurising Tolerance" := "Function ConditionCheck without valve"."Control B"."Time tolerance",
                           Pressurising_SP := "Function ConditionCheck without valve"."Input B".PressurisingSP,
                           Commissioning_mode := "Function ConditionCheck without valve"."Control B"."installation mode",
                           "Start ConditonCheck" := "Function ConditionCheck without valve"."Control B"."start Condition Check",
                           "Stop ConditonCheck" := "Function ConditionCheck without valve"."Control B"."stop Condition Check",
                           "ConditonCheck Running" := "Function ConditionCheck without valve"."Control B"."Condition Check running",
                           "ConditonCheck completed" := "Function ConditionCheck without valve"."Control B"."Condition Check Completed",
                           "ON Gear Pump" := "Function ConditionCheck without valve"."Output B"."ON pump",
                           "ON inlet" := "Function ConditionCheck without valve"."Output B"."ON_inlet B",
                           "dispensing Time PV" => "Function ConditionCheck without valve"."Output B"."running time",
                           "Checking Time pv" => "Function ConditionCheck without valve"."Output B".Pressure_release_time,
                           Leaktest_ok => "Function ConditionCheck without valve"."Output B".Pressure_OK,
                           Leaktest_nok => "Function ConditionCheck without valve"."Output B".Pressure_NOK,
                           Conditiontest_OK => "Function ConditionCheck without valve"."Output B"."Test Pass",
                           Conditiontest_NOK => "Function ConditionCheck without valve"."Output B".Test_Fail,
                           "PAT @ installation" => "Function ConditionCheck without valve"."Data B"."Pressure Achieved time @installation");
END_REGION

REGION Network 6
   RUNG wire#powerrail
      P_Contact(operand := "Function ConditionCheck without valve"."Control B"."installation mode", bit := "Temp".temp_4[6])
      S_Coil( "Function ConditionCheck without valve".reset_FIFOB )
   END_RUNG
   RUNG wire#powerrail
      Contact( "Function ConditionCheck without valve".reset_FIFOB )
      N_Contact(operand := "Functions"."1k"."Condition Check B", bit := "Temp".temp_4[4])
      R_Coil( "Function ConditionCheck without valve".reset_FIFOB )
   END_RUNG
   // the same network as SCL:
   #_w1 := "Function ConditionCheck without valve"."Control B"."installation mode" AND NOT "Temp".temp_4[6];   // rising edge of "Function ConditionCheck without valve"."Control B"."installation mode"
   "Temp".temp_4[6] := "Function ConditionCheck without valve"."Control B"."installation mode";
   IF #_w1 THEN "Function ConditionCheck without valve".reset_FIFOB := TRUE; END_IF;
   #_w2 := "Function ConditionCheck without valve".reset_FIFOB AND NOT "Functions"."1k"."Condition Check B" AND "Temp".temp_4[4];   // falling edge of "Functions"."1k"."Condition Check B"
   "Temp".temp_4[4] := "Functions"."1k"."Condition Check B";
   IF #_w2 THEN "Function ConditionCheck without valve".reset_FIFOB := FALSE; END_IF;
END_REGION

REGION Network 7
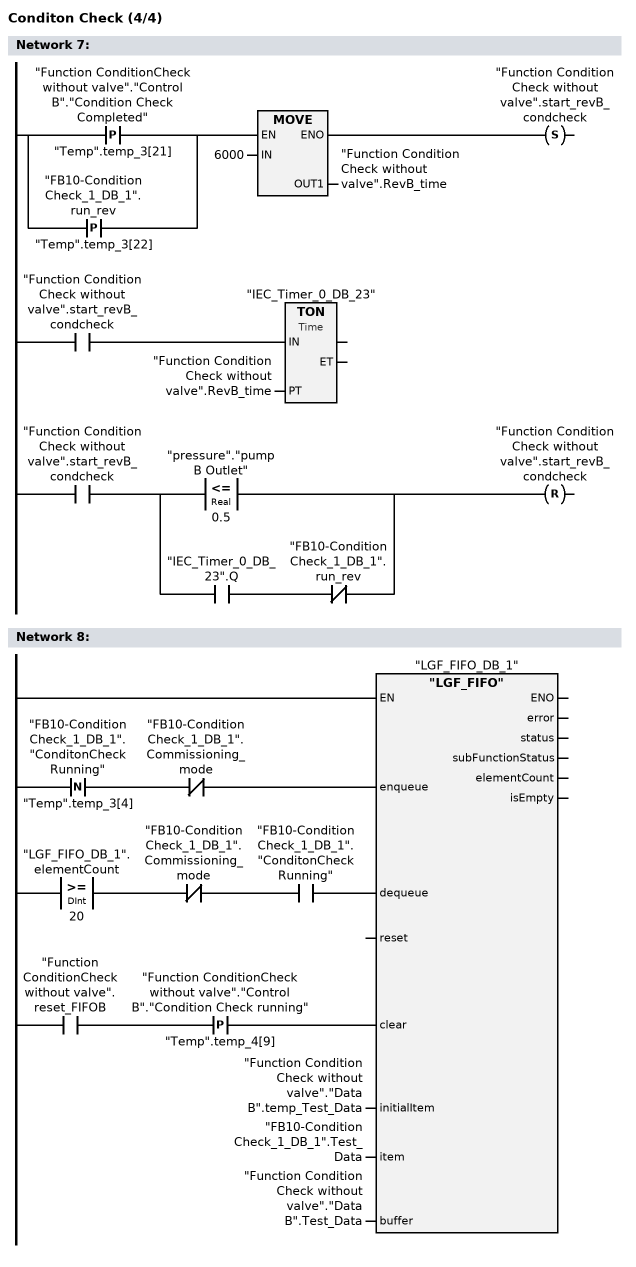
   RUNG wire#powerrail
      P_Contact(operand := "Function ConditionCheck without valve"."Control B"."Condition Check Completed", bit := "Temp".temp_3[21])
      wire#w1
      Move(in := 6000, out1 => "Function ConditionCheck without valve".RevB_time)
      S_Coil( "Function ConditionCheck without valve".start_revB_condcheck )
   END_RUNG
   RUNG wire#powerrail
      P_Contact(operand := "FB10-Condition Check_1_DB_1".run_rev, bit := "Temp".temp_3[22])
   END_RUNG wire#w1
   RUNG wire#powerrail
      Contact( "Function ConditionCheck without valve".start_revB_condcheck )
      { S7_Templates := "time_type := Time" } "IEC_Timer_0_DB_23".TON(pt := "Function ConditionCheck without valve".RevB_time, et =>)
   END_RUNG
   RUNG wire#powerrail
      Contact( "Function ConditionCheck without valve".start_revB_condcheck )
      wire#w2
      { S7_Templates := "SrcType := Real" } LE_Contact(in1 := "pressure"."pump B Outlet", in2 := 0.5)
      wire#w3
      R_Coil( "Function ConditionCheck without valve".start_revB_condcheck )
   END_RUNG
   RUNG wire#w2
      Contact( "IEC_Timer_0_DB_23".Q )
      I_Contact( "FB10-Condition Check_1_DB_1".run_rev )
   END_RUNG wire#w3
   // the same network as SCL:
   #_w1 := "Function ConditionCheck without valve"."Control B"."Condition Check Completed" AND NOT "Temp".temp_3[21];   // rising edge of "Function ConditionCheck without valve"."Control B"."Condition Check Completed"
   "Temp".temp_3[21] := "Function ConditionCheck without valve"."Control B"."Condition Check Completed";
   #_w2 := "FB10-Condition Check_1_DB_1".run_rev AND NOT "Temp".temp_3[22];   // rising edge of "FB10-Condition Check_1_DB_1".run_rev
   "Temp".temp_3[22] := "FB10-Condition Check_1_DB_1".run_rev;
   IF #_w1 OR #_w2 THEN
       "Function ConditionCheck without valve".RevB_time := 6000;
       "Function ConditionCheck without valve".start_revB_condcheck := TRUE;
   END_IF;
   "IEC_Timer_0_DB_23".TON(IN := "Function ConditionCheck without valve".start_revB_condcheck,
                           PT := "Function ConditionCheck without valve".RevB_time);
   IF "Function ConditionCheck without valve".start_revB_condcheck AND (("pressure"."pump B Outlet" <= 0.5) OR ("IEC_Timer_0_DB_23".Q AND NOT "FB10-Condition Check_1_DB_1".run_rev)) THEN
       "Function ConditionCheck without valve".start_revB_condcheck := FALSE;
   END_IF;
END_REGION

REGION Network 8
   RUNG wire#powerrail
      "LGF_FIFO_DB_1"(enqueue := wire#w1, dequeue := wire#w2, clear := wire#w3, reset :=, initialItem := "Function ConditionCheck without valve"."Data B".temp_Test_Data, item := "FB10-Condition Check_1_DB_1".Test_Data, buffer := "Function ConditionCheck without valve"."Data B".Test_Data, error =>, status =>, subFunctionStatus =>, elementCount =>, isEmpty =>)
   END_RUNG
   RUNG wire#powerrail
      N_Contact(operand := "FB10-Condition Check_1_DB_1"."ConditonCheck Running", bit := "Temp".temp_3[4])
      I_Contact( "FB10-Condition Check_1_DB_1".Commissioning_mode )
   END_RUNG wire#w1
   RUNG wire#powerrail
      { S7_Templates := "SrcType := DInt" } GE_Contact(in1 := "LGF_FIFO_DB_1".elementCount, in2 := 20)
      I_Contact( "FB10-Condition Check_1_DB_1".Commissioning_mode )
      Contact( "FB10-Condition Check_1_DB_1"."ConditonCheck Running" )
   END_RUNG wire#w2
   RUNG wire#powerrail
      Contact( "Function ConditionCheck without valve".reset_FIFOB )
      P_Contact(operand := "Function ConditionCheck without valve"."Control B"."Condition Check running", bit := "Temp".temp_4[9])
   END_RUNG wire#w3
   // the same network as SCL:
   #_w1 := NOT "FB10-Condition Check_1_DB_1"."ConditonCheck Running" AND "Temp".temp_3[4];   // falling edge of "FB10-Condition Check_1_DB_1"."ConditonCheck Running"
   "Temp".temp_3[4] := "FB10-Condition Check_1_DB_1"."ConditonCheck Running";
   #_w2 := "Function ConditionCheck without valve".reset_FIFOB AND "Function ConditionCheck without valve"."Control B"."Condition Check running" AND NOT "Temp".temp_4[9];   // rising edge of "Function ConditionCheck without valve"."Control B"."Condition Check running"
   "Temp".temp_4[9] := "Function ConditionCheck without valve"."Control B"."Condition Check running";
   "LGF_FIFO_DB_1"(enqueue := #_w1 AND NOT "FB10-Condition Check_1_DB_1".Commissioning_mode,   // "LGF_FIFO"
                   dequeue := ("LGF_FIFO_DB_1".elementCount >= 20) AND NOT "FB10-Condition Check_1_DB_1".Commissioning_mode AND "FB10-Condition Check_1_DB_1"."ConditonCheck Running",
                   clear := #_w2,
                   initialItem := "Function ConditionCheck without valve"."Data B".temp_Test_Data,
                   item := "FB10-Condition Check_1_DB_1".Test_Data,
                   buffer := "Function ConditionCheck without valve"."Data B".Test_Data);
END_REGION
END_FUNCTION

FUNCTION_BLOCK "FB10-Condition Check_1"   // FB14, LAD
{ S7_Optimized_Access := 'TRUE' }
VERSION : 0.1
// stored: AutoNumber true, IsIECCheckEnabled false, IsRetainMemResEnabled false, MemoryReserve 100, SetENOAutomatically false, UDAEnableTagReadback false
   VAR_INPUT
      "Time" : DInt;
      "Pump ON delay" : DInt;
      Check_Time { ExternalAccessible := 'False'; ExternalVisible := 'False'; ExternalWritable := 'False'} : DInt;
      Pressure_SP { ExternalAccessible := 'False'; ExternalVisible := 'False'; ExternalWritable := 'False'} : Real;
      Pressure_tolerance { ExternalAccessible := 'False'; ExternalVisible := 'False'; ExternalWritable := 'False'} : Real;
      Current_pressure { ExternalAccessible := 'False'; ExternalVisible := 'False'; ExternalWritable := 'False'} : Real;
      selected { ExternalAccessible := 'False'; ExternalVisible := 'False'; ExternalWritable := 'False'} : Bool;
      "Pressurising Tolerance" : Real;
      Pressurising_SP : Real;
   END_VAR
   VAR_OUTPUT
      "dispensing Time PV" : Int;
      "Checking Time pv" { ExternalAccessible := 'False'; ExternalVisible := 'False'; ExternalWritable := 'False'} : Int;
      Leaktest_ok { ExternalAccessible := 'False'; ExternalVisible := 'False'; ExternalWritable := 'False'} : Bool;
      Leaktest_nok { ExternalAccessible := 'False'; ExternalVisible := 'False'; ExternalWritable := 'False'} : Bool;
      Conditiontest_OK : Bool;
      Conditiontest_NOK { ExternalAccessible := 'False'; ExternalVisible := 'False'; ExternalWritable := 'False'} : Bool;
      "PAT @ installation" : DInt;   // Pressure achieved Time @ Installation
      Test_Data : "Condition_Check";
   END_VAR
   VAR_IN_OUT
      Commissioning_mode : Bool;
      "Start ConditonCheck" : Bool;
      "Stop ConditonCheck" : Bool;
      "ConditonCheck Running" : Bool;
      "ConditonCheck completed" : Bool;
      "ON Gear Pump" : Bool;
      "ON inlet" : Bool;
      Pressurising : Bool;
      run_rev : Bool;
   END_VAR
   VAR
      "dispensing time done" : Bool;
      "dispensing time in sec" : DInt;
      "timer input" : DInt;
      IEC_Timer_0_Instance_1 { S7_SetPoint := 'True'} : TON_TIME;
      IEC_Timer_0_Instance_2 { S7_SetPoint := 'True'} : TON_TIME;
      IEC_Timer_0_Instance_4 { S7_SetPoint := 'True'} : TON_TIME;
      "Press+ve" { ExternalAccessible := 'False'; ExternalVisible := 'False'; ExternalWritable := 'False'; S7_SetPoint := 'True'} : Real;
      "Press-ve" { ExternalAccessible := 'False'; ExternalVisible := 'False'; ExternalWritable := 'False'} : Real;
      IEC_Timer_0_Instance_3 { ExternalAccessible := 'False'; ExternalVisible := 'False'; ExternalWritable := 'False'; S7_SetPoint := 'True'} : TON_TIME;
      Checktime_ms { ExternalAccessible := 'False'; ExternalVisible := 'False'; ExternalWritable := 'False'; S7_SetPoint := 'True'} : DInt;
      Check_timesec { ExternalAccessible := 'False'; ExternalVisible := 'False'; ExternalWritable := 'False'} : DInt;
      temp_ons { ExternalAccessible := 'False'; ExternalVisible := 'False'; ExternalWritable := 'False'} : Bool;
      temp : Array[0..5] of Bool;
      IEC_Timer_0_Instance_5 { S7_SetPoint := 'True'} : TON_TIME;
      "WIth Tolerance" { S7_SetPoint := 'True'} : DInt;
      Pressure_achive_time : DInt;
      Pressure_ok : Bool;
      IEC_Timer_0_Instance { S7_SetPoint := 'True'} : TON_TIME;
      Result { S7_SetPoint := 'True'} : Bool;
      "result temp" : Bool;
      IEC_Timer_0_Instance_6 { S7_SetPoint := 'True'} : TON_TIME;
      Start_cond : Bool;
      IEC_Timer_0_Instance_7 { S7_SetPoint := 'True'} : TON_TIME;
   END_VAR
   VAR_TEMP
      ret : Int;
   END_VAR
   VAR_TEMP   // added for the SCL form of the ladder/FBD networks
      _w1 : Bool;
      _w2 : Bool;
      _w3 : Bool;
      _w4 : Bool;
      _w5 : Bool;
   END_VAR
BEGIN

REGION Network 1
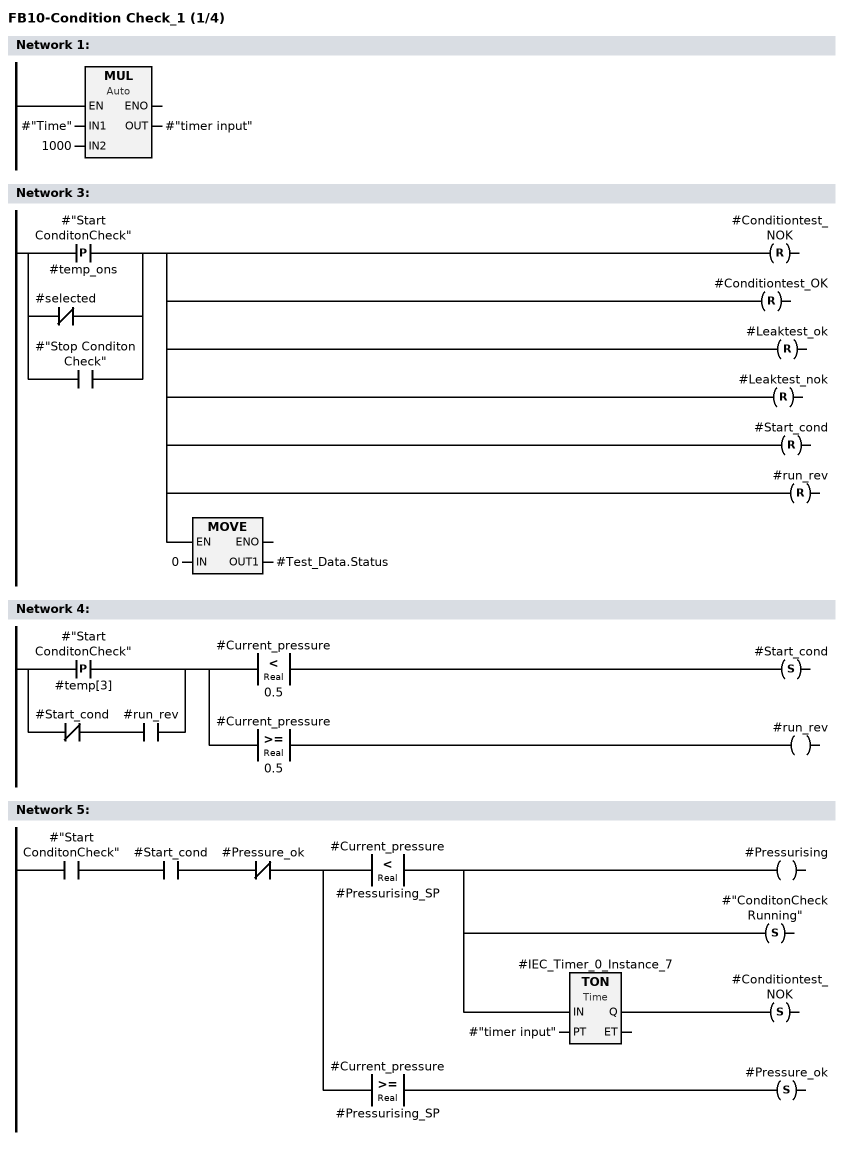
   RUNG wire#powerrail
      Mul(in1 := #"Time", in2 := 1000, out => #"timer input")
   END_RUNG
   // the same network as SCL:
   #"timer input" := #"Time" * 1000;
END_REGION

REGION Network 2 (SCL)
   #"WIth Tolerance" := ROUND(#"PAT @ installation" + ((#"PAT @ installation"*#"Pressurising Tolerance")/100));
END_REGION

REGION Network 3
   RUNG wire#powerrail
      P_Contact(operand := #"Start ConditonCheck", bit := #temp_ons)
      wire#w1
      R_Coil( #Conditiontest_NOK )
   END_RUNG
   RUNG wire#powerrail
      I_Contact( #selected )
   END_RUNG wire#w1
   RUNG wire#powerrail
      Contact( #"Stop ConditonCheck" )
   END_RUNG wire#w1
   RUNG wire#w1
      R_Coil( #Conditiontest_OK )
   END_RUNG
   RUNG wire#w1
      R_Coil( #Leaktest_ok )
   END_RUNG
   RUNG wire#w1
      R_Coil( #Leaktest_nok )
   END_RUNG
   RUNG wire#w1
      R_Coil( #Start_cond )
   END_RUNG
   RUNG wire#w1
      R_Coil( #run_rev )
   END_RUNG
   RUNG wire#w1
      Move(in := 0, out1 => #Test_Data.Status)
   END_RUNG
   // the same network as SCL:
   #_w1 := #"Start ConditonCheck" AND NOT #temp_ons;   // rising edge of #"Start ConditonCheck"
   #temp_ons := #"Start ConditonCheck";
   IF #_w1 OR NOT #selected OR #"Stop ConditonCheck" THEN
       #Conditiontest_NOK := FALSE;
       #Conditiontest_OK := FALSE;
       #Leaktest_ok := FALSE;
       #Leaktest_nok := FALSE;
       #Start_cond := FALSE;
       #run_rev := FALSE;
       #Test_Data.Status := 0;
   END_IF;
END_REGION

REGION Network 4
   RUNG wire#powerrail
      P_Contact(operand := #"Start ConditonCheck", bit := #temp[3])
      wire#w1
      { S7_Templates := "SrcType := Real" } LT_Contact(in1 := #Current_pressure, in2 := 0.5)
      S_Coil( #Start_cond )
   END_RUNG
   RUNG wire#powerrail
      I_Contact( #Start_cond )
      Contact( #run_rev )
   END_RUNG wire#w1
   RUNG wire#w1
      { S7_Templates := "SrcType := Real" } GE_Contact(in1 := #Current_pressure, in2 := 0.5)
      Coil( #run_rev )
   END_RUNG
   // the same network as SCL:
   #_w1 := #"Start ConditonCheck" AND NOT #temp[3];   // rising edge of #"Start ConditonCheck"
   #temp[3] := #"Start ConditonCheck";
   #_w2 := #_w1 OR (NOT #Start_cond AND #run_rev);
   IF #_w2 AND (#Current_pressure < 0.5) THEN #Start_cond := TRUE; END_IF;
   #run_rev := #_w2 AND (#Current_pressure >= 0.5);
END_REGION

REGION Network 5
   RUNG wire#powerrail
      Contact( #"Start ConditonCheck" )
      Contact( #Start_cond )
      I_Contact( #Pressure_ok )
      wire#w1
      { S7_Templates := "SrcType := Real" } LT_Contact(in1 := #Current_pressure, in2 := #Pressurising_SP)
      wire#w2
      Coil( #Pressurising )
   END_RUNG
   RUNG wire#w2
      S_Coil( #"ConditonCheck Running" )
   END_RUNG
   RUNG wire#w2
      { S7_Templates := "time_type := Time" } #IEC_Timer_0_Instance_7.TON(pt := #"timer input", et =>)
      S_Coil( #Conditiontest_NOK )
   END_RUNG
   RUNG wire#w1
      { S7_Templates := "SrcType := Real" } GE_Contact(in1 := #Current_pressure, in2 := #Pressurising_SP)
      S_Coil( #Pressure_ok )
   END_RUNG
   // the same network as SCL:
   #_w1 := #"Start ConditonCheck" AND #Start_cond AND NOT #Pressure_ok;
   #Pressurising := #_w1 AND (#Current_pressure < #Pressurising_SP);
   IF #Pressurising THEN #"ConditonCheck Running" := TRUE; END_IF;
   #IEC_Timer_0_Instance_7(IN := #Pressurising, PT := #"timer input");   // TON
   IF #IEC_Timer_0_Instance_7.Q THEN #Conditiontest_NOK := TRUE; END_IF;
   IF #_w1 AND (#Current_pressure >= #Pressurising_SP) THEN #Pressure_ok := TRUE; END_IF;
END_REGION

REGION Network 6
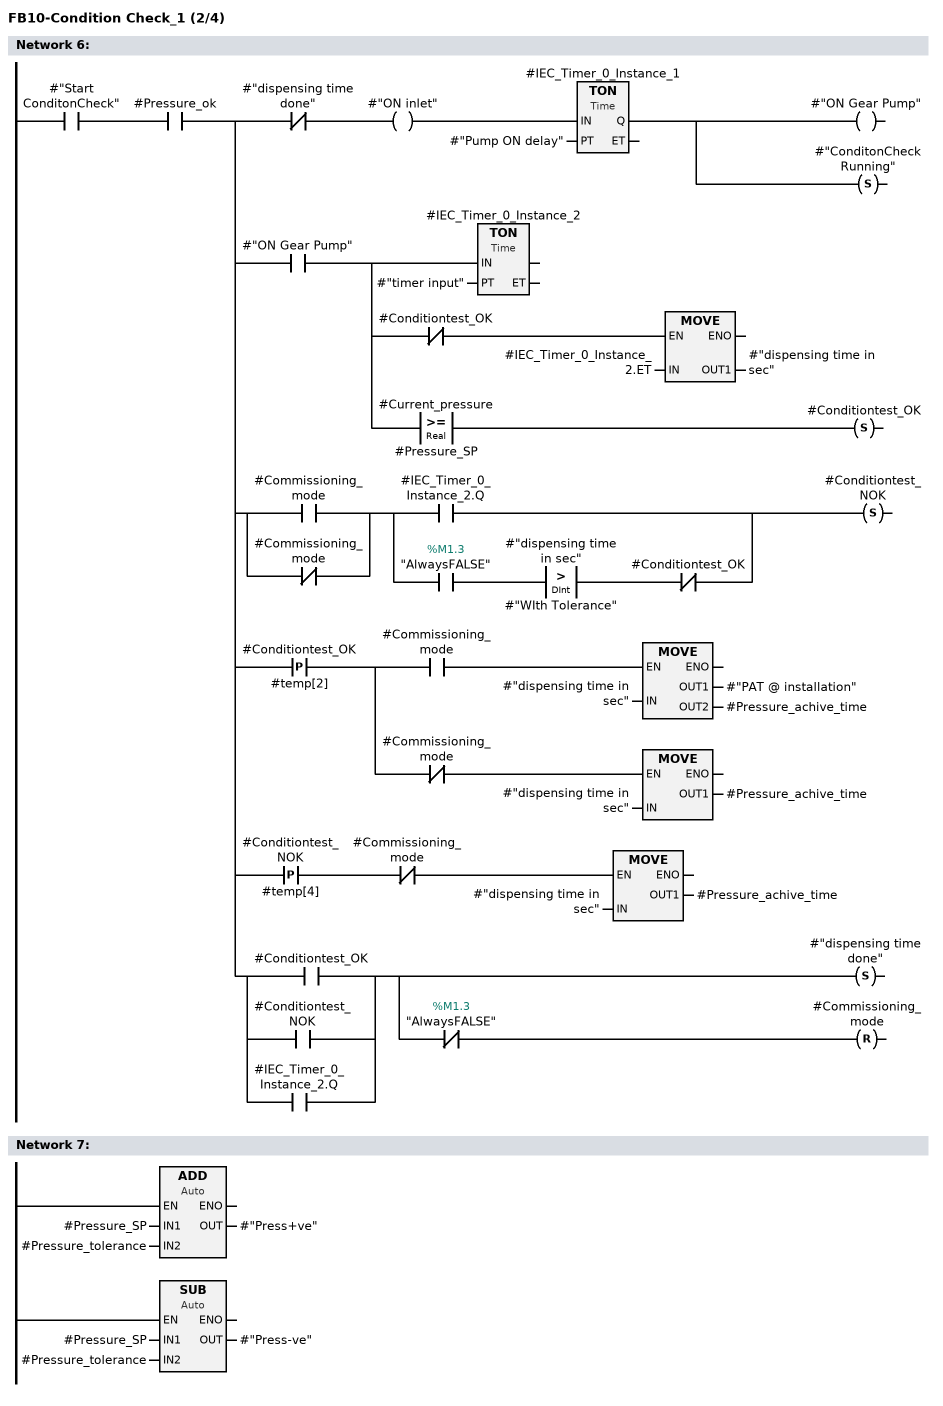
   RUNG wire#powerrail
      Contact( #"Start ConditonCheck" )
      Contact( #Pressure_ok )
      wire#w1
      I_Contact( #"dispensing time done" )
      Coil( #"ON inlet" )
      { S7_Templates := "time_type := Time" } #IEC_Timer_0_Instance_1.TON(pt := #"Pump ON delay", et =>)
      wire#w2
      Coil( #"ON Gear Pump" )
   END_RUNG
   RUNG wire#w2
      S_Coil( #"ConditonCheck Running" )
   END_RUNG
   RUNG wire#w1
      Contact( #"ON Gear Pump" )
      wire#w3
      { S7_Templates := "time_type := Time" } #IEC_Timer_0_Instance_2.TON(pt := #"timer input", et =>)
   END_RUNG
   RUNG wire#w3
      I_Contact( #Conditiontest_OK )
      Move(in := #IEC_Timer_0_Instance_2.ET, out1 => #"dispensing time in sec")
   END_RUNG
   RUNG wire#w3
      { S7_Templates := "SrcType := Real" } GE_Contact(in1 := #Current_pressure, in2 := #Pressure_SP)
      S_Coil( #Conditiontest_OK )
   END_RUNG
   RUNG wire#w1
      Contact( #Commissioning_mode )
      wire#w4
      Contact( #IEC_Timer_0_Instance_2.Q )
      wire#w5
      S_Coil( #Conditiontest_NOK )
   END_RUNG
   RUNG wire#w1
      I_Contact( #Commissioning_mode )
   END_RUNG wire#w4
   RUNG wire#w4
      Contact( "AlwaysFALSE" )
      { S7_Templates := "SrcType := DInt" } GT_Contact(in1 := #"dispensing time in sec", in2 := #"WIth Tolerance")
      I_Contact( #Conditiontest_OK )
   END_RUNG wire#w5
   RUNG wire#w1
      P_Contact(operand := #Conditiontest_OK, bit := #temp[2])
      wire#w6
      Contact( #Commissioning_mode )
      Move(in := #"dispensing time in sec", out1 => #"PAT @ installation", out2 => #Pressure_achive_time)
   END_RUNG
   RUNG wire#w6
      I_Contact( #Commissioning_mode )
      Move(in := #"dispensing time in sec", out1 => #Pressure_achive_time)
   END_RUNG
   RUNG wire#w1
      P_Contact(operand := #Conditiontest_NOK, bit := #temp[4])
      I_Contact( #Commissioning_mode )
      Move(in := #"dispensing time in sec", out1 => #Pressure_achive_time)
   END_RUNG
   RUNG wire#w1
      Contact( #Conditiontest_OK )
      wire#w7
      S_Coil( #"dispensing time done" )
   END_RUNG
   RUNG wire#w1
      Contact( #Conditiontest_NOK )
   END_RUNG wire#w7
   RUNG wire#w1
      Contact( #IEC_Timer_0_Instance_2.Q )
   END_RUNG wire#w7
   RUNG wire#w7
      I_Contact( "AlwaysFALSE" )
      R_Coil( #Commissioning_mode )
   END_RUNG
   // the same network as SCL:
   #_w1 := #"Start ConditonCheck" AND #Pressure_ok;
   #"ON inlet" := #_w1 AND NOT #"dispensing time done";
   #IEC_Timer_0_Instance_1(IN := #"ON inlet", PT := #"Pump ON delay");   // TON
   #"ON Gear Pump" := #IEC_Timer_0_Instance_1.Q;
   IF #IEC_Timer_0_Instance_1.Q THEN #"ConditonCheck Running" := TRUE; END_IF;
   #_w2 := #_w1 AND #"ON Gear Pump";
   #IEC_Timer_0_Instance_2(IN := #_w2, PT := #"timer input");   // TON
   IF #_w2 AND NOT #Conditiontest_OK THEN #"dispensing time in sec" := #IEC_Timer_0_Instance_2.ET; END_IF;
   IF #_w2 AND (#Current_pressure >= #Pressure_SP) THEN #Conditiontest_OK := TRUE; END_IF;
   IF #_w1 AND (#Commissioning_mode OR NOT #Commissioning_mode) AND (#IEC_Timer_0_Instance_2.Q OR ("AlwaysFALSE" AND (#"dispensing time in sec" > #"WIth Tolerance") AND NOT #Conditiontest_OK)) THEN
       #Conditiontest_NOK := TRUE;
   END_IF;
   #_w3 := #_w1 AND #Conditiontest_OK AND NOT #temp[2];   // rising edge of #Conditiontest_OK
   #temp[2] := #Conditiontest_OK;
   IF #_w3 AND #Commissioning_mode THEN
       #"PAT @ installation" := #"dispensing time in sec";
       #Pressure_achive_time := #"dispensing time in sec";
   END_IF;
   IF #_w3 AND NOT #Commissioning_mode THEN #Pressure_achive_time := #"dispensing time in sec"; END_IF;
   #_w4 := #_w1 AND #Conditiontest_NOK AND NOT #temp[4];   // rising edge of #Conditiontest_NOK
   #temp[4] := #Conditiontest_NOK;
   IF #_w4 AND NOT #Commissioning_mode THEN #Pressure_achive_time := #"dispensing time in sec"; END_IF;
   #_w5 := #_w1 AND (#Conditiontest_OK OR #Conditiontest_NOK OR #IEC_Timer_0_Instance_2.Q);
   IF #_w5 THEN #"dispensing time done" := TRUE; END_IF;
   IF #_w5 AND NOT "AlwaysFALSE" THEN #Commissioning_mode := FALSE; END_IF;
END_REGION

REGION Network 7
   RUNG wire#powerrail
      Add(in1 := #Pressure_SP, in2 := #Pressure_tolerance, out => #"Press+ve")
   END_RUNG
   RUNG wire#powerrail
      Sub(in1 := #Pressure_SP, in2 := #Pressure_tolerance, out => #"Press-ve")
   END_RUNG
   // the same network as SCL:
   #"Press+ve" := #Pressure_SP + #Pressure_tolerance;
   #"Press-ve" := #Pressure_SP - #Pressure_tolerance;
END_REGION

REGION Network 8
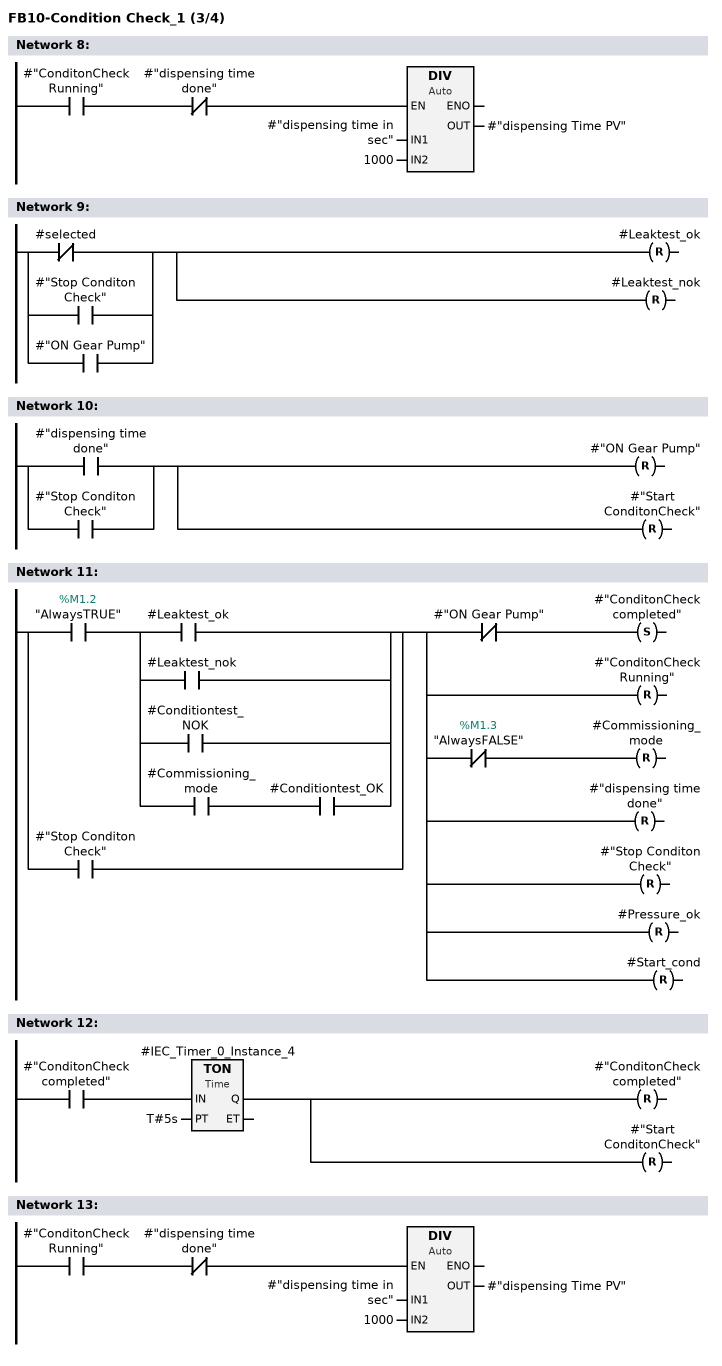
   RUNG wire#powerrail
      Contact( #"ConditonCheck Running" )
      I_Contact( #"dispensing time done" )
      Div(in1 := #"dispensing time in sec", in2 := 1000, out => #"dispensing Time PV")
   END_RUNG
   // the same network as SCL:
   IF #"ConditonCheck Running" AND NOT #"dispensing time done" THEN
       #"dispensing Time PV" := #"dispensing time in sec" / 1000;
   END_IF;
END_REGION

REGION Network 9
   RUNG wire#powerrail
      I_Contact( #selected )
      wire#w1
      R_Coil( #Leaktest_ok )
   END_RUNG
   RUNG wire#powerrail
      Contact( #"Stop ConditonCheck" )
   END_RUNG wire#w1
   RUNG wire#powerrail
      Contact( #"ON Gear Pump" )
   END_RUNG wire#w1
   RUNG wire#w1
      R_Coil( #Leaktest_nok )
   END_RUNG
   // the same network as SCL:
   IF NOT #selected OR #"Stop ConditonCheck" OR #"ON Gear Pump" THEN
       #Leaktest_ok := FALSE;
       #Leaktest_nok := FALSE;
   END_IF;
END_REGION

REGION Network 10
   RUNG wire#powerrail
      Contact( #"dispensing time done" )
      wire#w1
      R_Coil( #"ON Gear Pump" )
   END_RUNG
   RUNG wire#powerrail
      Contact( #"Stop ConditonCheck" )
   END_RUNG wire#w1
   RUNG wire#w1
      R_Coil( #"Start ConditonCheck" )
   END_RUNG
   // the same network as SCL:
   IF #"dispensing time done" OR #"Stop ConditonCheck" THEN
       #"ON Gear Pump" := FALSE;
       #"Start ConditonCheck" := FALSE;
   END_IF;
END_REGION

REGION Network 11
   RUNG wire#powerrail
      Contact( "AlwaysTRUE" )
      wire#w1
      Contact( #Leaktest_ok )
      wire#w2
      I_Contact( #"ON Gear Pump" )
      S_Coil( #"ConditonCheck completed" )
   END_RUNG
   RUNG wire#w1
      Contact( #Leaktest_nok )
   END_RUNG wire#w2
   RUNG wire#w1
      Contact( #Conditiontest_NOK )
   END_RUNG wire#w2
   RUNG wire#w1
      Contact( #Commissioning_mode )
      Contact( #Conditiontest_OK )
   END_RUNG wire#w2
   RUNG wire#powerrail
      Contact( #"Stop ConditonCheck" )
   END_RUNG wire#w2
   RUNG wire#w2
      R_Coil( #"ConditonCheck Running" )
   END_RUNG
   RUNG wire#w2
      I_Contact( "AlwaysFALSE" )
      R_Coil( #Commissioning_mode )
   END_RUNG
   RUNG wire#w2
      R_Coil( #"dispensing time done" )
   END_RUNG
   RUNG wire#w2
      R_Coil( #"Stop ConditonCheck" )
   END_RUNG
   RUNG wire#w2
      R_Coil( #Pressure_ok )
   END_RUNG
   RUNG wire#w2
      R_Coil( #Start_cond )
   END_RUNG
   // the same network as SCL:
   #_w1 := ("AlwaysTRUE" AND (#Leaktest_ok OR #Leaktest_nok OR #Conditiontest_NOK OR (#Commissioning_mode AND #Conditiontest_OK))) OR #"Stop ConditonCheck";
   IF #_w1 AND NOT #"ON Gear Pump" THEN #"ConditonCheck completed" := TRUE; END_IF;
   IF #_w1 THEN #"ConditonCheck Running" := FALSE; END_IF;
   IF #_w1 AND NOT "AlwaysFALSE" THEN #Commissioning_mode := FALSE; END_IF;
   IF #_w1 THEN
       #"dispensing time done" := FALSE;
       #"Stop ConditonCheck" := FALSE;
       #Pressure_ok := FALSE;
       #Start_cond := FALSE;
   END_IF;
END_REGION

REGION Network 12
   RUNG wire#powerrail
      Contact( #"ConditonCheck completed" )
      { S7_Templates := "time_type := Time" } #IEC_Timer_0_Instance_4.TON(pt := T#5s, et =>)
      wire#w1
      R_Coil( #"ConditonCheck completed" )
   END_RUNG
   RUNG wire#w1
      R_Coil( #"Start ConditonCheck" )
   END_RUNG
   // the same network as SCL:
   #IEC_Timer_0_Instance_4(IN := #"ConditonCheck completed", PT := T#5s);   // TON
   IF #IEC_Timer_0_Instance_4.Q THEN
       #"ConditonCheck completed" := FALSE;
       #"Start ConditonCheck" := FALSE;
   END_IF;
END_REGION

REGION Network 13
   RUNG wire#powerrail
      Contact( #"ConditonCheck Running" )
      I_Contact( #"dispensing time done" )
      Div(in1 := #"dispensing time in sec", in2 := 1000, out => #"dispensing Time PV")
   END_RUNG
   // the same network as SCL:
   IF #"ConditonCheck Running" AND NOT #"dispensing time done" THEN
       #"dispensing Time PV" := #"dispensing time in sec" / 1000;
   END_IF;
END_REGION

REGION Network 14
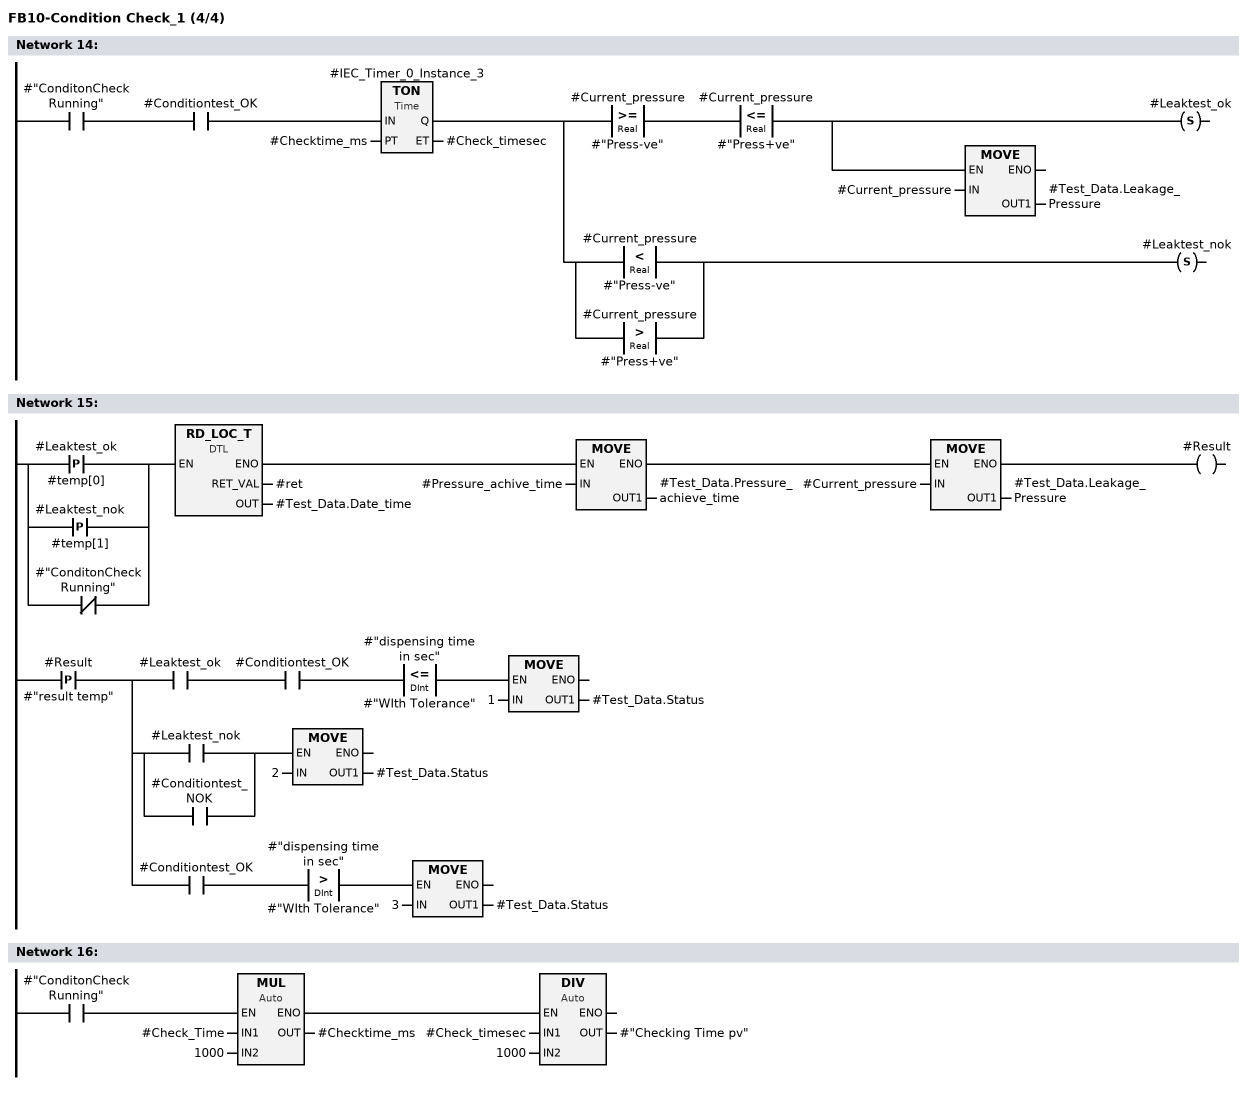
   RUNG wire#powerrail
      Contact( #"ConditonCheck Running" )
      Contact( #Conditiontest_OK )
      { S7_Templates := "time_type := Time" } #IEC_Timer_0_Instance_3.TON(pt := #Checktime_ms, et => #Check_timesec)
      wire#w1
      { S7_Templates := "SrcType := Real" } GE_Contact(in1 := #Current_pressure, in2 := #"Press-ve")
      { S7_Templates := "SrcType := Real" } LE_Contact(in1 := #Current_pressure, in2 := #"Press+ve")
      wire#w2
      S_Coil( #Leaktest_ok )
   END_RUNG
   RUNG wire#w2
      Move(in := #Current_pressure, out1 => #Test_Data.Leakage_Pressure)
   END_RUNG
   RUNG wire#w1
      { S7_Templates := "SrcType := Real" } LT_Contact(in1 := #Current_pressure, in2 := #"Press-ve")
      wire#w3
      S_Coil( #Leaktest_nok )
   END_RUNG
   RUNG wire#w1
      { S7_Templates := "SrcType := Real" } GT_Contact(in1 := #Current_pressure, in2 := #"Press+ve")
   END_RUNG wire#w3
   // the same network as SCL:
   #IEC_Timer_0_Instance_3(IN := #"ConditonCheck Running" AND #Conditiontest_OK,   // TON
                           PT := #Checktime_ms,
                           ET => #Check_timesec);
   IF #IEC_Timer_0_Instance_3.Q AND (#Current_pressure >= #"Press-ve") AND (#Current_pressure <= #"Press+ve") THEN
       #Leaktest_ok := TRUE;
       #Test_Data.Leakage_Pressure := #Current_pressure;
   END_IF;
   IF #IEC_Timer_0_Instance_3.Q AND ((#Current_pressure < #"Press-ve") OR (#Current_pressure > #"Press+ve")) THEN
       #Leaktest_nok := TRUE;
   END_IF;
END_REGION

REGION Network 15
   RUNG wire#powerrail
      P_Contact(operand := #Leaktest_ok, bit := #temp[0])
      wire#w1
      { S7_Templates := "date_type := DTL" } RD_LOC_T(RET_VAL => #ret, OUT => #Test_Data.Date_time)
      Move(in := #Pressure_achive_time, out1 => #Test_Data.Pressure_achieve_time)
      Move(in := #Current_pressure, out1 => #Test_Data.Leakage_Pressure)
      Coil( #Result )
   END_RUNG
   RUNG wire#powerrail
      P_Contact(operand := #Leaktest_nok, bit := #temp[1])
   END_RUNG wire#w1
   RUNG wire#powerrail
      I_Contact( #"ConditonCheck Running" )
   END_RUNG wire#w1
   RUNG wire#powerrail
      P_Contact(operand := #Result, bit := #"result temp")
      wire#w2
      Contact( #Leaktest_ok )
      Contact( #Conditiontest_OK )
      { S7_Templates := "SrcType := DInt" } LE_Contact(in1 := #"dispensing time in sec", in2 := #"WIth Tolerance")
      Move(in := 1, out1 => #Test_Data.Status)
   END_RUNG
   RUNG wire#w2
      Contact( #Leaktest_nok )
      wire#w3
      Move(in := 2, out1 => #Test_Data.Status)
   END_RUNG
   RUNG wire#w2
      Contact( #Conditiontest_NOK )
   END_RUNG wire#w3
   RUNG wire#w2
      Contact( #Conditiontest_OK )
      { S7_Templates := "SrcType := DInt" } GT_Contact(in1 := #"dispensing time in sec", in2 := #"WIth Tolerance")
      Move(in := 3, out1 => #Test_Data.Status)
   END_RUNG
   // the same network as SCL:
   #_w1 := #Leaktest_ok AND NOT #temp[0];   // rising edge of #Leaktest_ok
   #temp[0] := #Leaktest_ok;
   #_w2 := #Leaktest_nok AND NOT #temp[1];   // rising edge of #Leaktest_nok
   #temp[1] := #Leaktest_nok;
   #_w3 := #_w1 OR #_w2 OR NOT #"ConditonCheck Running";
   #ret := RD_LOC_T(EN := #_w3, OUT => #Test_Data.Date_time, ENO => #_w4);
   IF #_w4 THEN
       #Test_Data.Pressure_achieve_time := #Pressure_achive_time;
       #Test_Data.Leakage_Pressure := #Current_pressure;
   END_IF;
   #Result := #_w4;
   #_w5 := #Result AND NOT #"result temp";   // rising edge of #Result
   #"result temp" := #Result;
   IF #_w5 AND #Leaktest_ok AND #Conditiontest_OK AND (#"dispensing time in sec" <= #"WIth Tolerance") THEN
       #Test_Data.Status := 1;
   END_IF;
   IF #_w5 AND (#Leaktest_nok OR #Conditiontest_NOK) THEN #Test_Data.Status := 2; END_IF;
   IF #_w5 AND #Conditiontest_OK AND (#"dispensing time in sec" > #"WIth Tolerance") THEN
       #Test_Data.Status := 3;
   END_IF;
END_REGION

REGION Network 16
   RUNG wire#powerrail
      Contact( #"ConditonCheck Running" )
      Mul(in1 := #Check_Time, in2 := 1000, out => #Checktime_ms)
      Div(in1 := #Check_timesec, in2 := 1000, out => #"Checking Time pv")
   END_RUNG
   // the same network as SCL:
   IF #"ConditonCheck Running" THEN
       #Checktime_ms := #Check_Time * 1000;
       #"Checking Time pv" := #Check_timesec / 1000;
   END_IF;
END_REGION
END_FUNCTION_BLOCK

FUNCTION "MR_Quantity Control" : Void   // FC16, LAD
{ S7_Optimized_Access := 'TRUE' }
VERSION : 0.1
// stored: AutoNumber true, IsIECCheckEnabled false, SetENOAutomatically false, UDAEnableTagReadback false
   VAR_TEMP
      temp : Bool;
   END_VAR
BEGIN

REGION Network 1 (SCL)
       //IF "Function Ratio check".input.Mode = 0 THEN
           "Function Ratio check".PumpCaliberationControls.CurrentSet_A := (100 / ("Mixing ratio"."Mixing ratio according to density" + real#100)) * "Function Ratio check".input."set qty";
         "Function Ratio check".PumpCaliberationControls.CurrentSet_B := "Function Ratio check".input."set qty" - "Function Ratio check".PumpCaliberationControls.CurrentSet_A;
      // END_IF;

       // IF "Function Ratio check".input.Mode = 1 THEN
       //     "Function Ratio check".PumpCaliberationControls.CurrentSet_A := "Function Ratio check".input."set qty";
       //    // "Function Ratio check".PumpCaliberationControls.CurrentSet_B := 0;
       //   //"Function Ratio check".PumpCaliberationControls.CurrentSet_B := "Function Ratio check".input."set qty" - "Function Ratio check".PumpCaliberationControls.CurrentSet_A;
       // END_IF;

       // IF "Function Ratio check".input.Mode = 2 THEN
       //  // "Function Ratio check".PumpCaliberationControls.CurrentSet_A := 0;
       //   "Function Ratio check".PumpCaliberationControls.CurrentSet_B := "Function Ratio check".input."set qty";//- "Function Ratio check".PumpCaliberationControls.CurrentSet_A;
       // END_IF;


       //Progress bar Higher limit for Ratio check to display on the screen.
       "Function Ratio check".Control.ProgressBar_Limit := REAL_TO_DINT(("Function Ratio check".input."set qty" / "Function Ratio check".input."Set Flowrate") * 60000);

       // Actual progress bar display on the screen for Ratio check progress.
       "Function Ratio check".Control.ProgressBar := "Function Ratio check".output."Running time" * 1000;
END_REGION

REGION Network 2
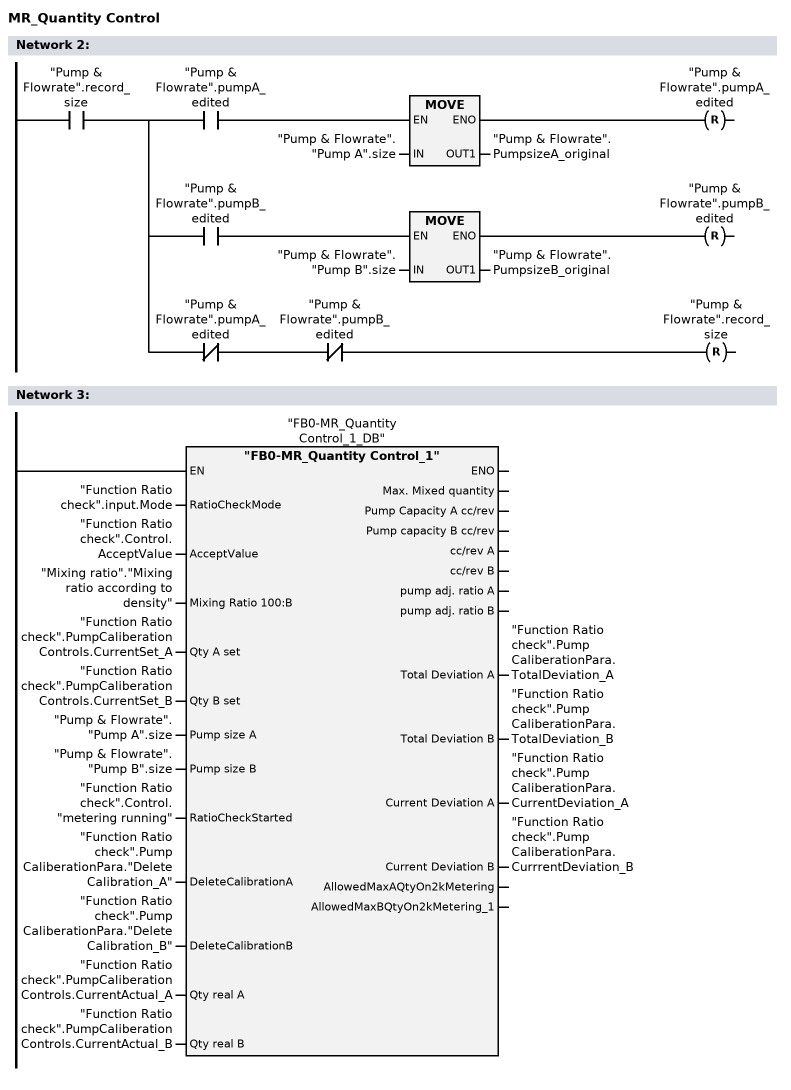
   IF "Pump & Flowrate".record_size AND "Pump & Flowrate".pumpA_edited THEN
       "Pump & Flowrate".PumpsizeA_original := "Pump & Flowrate"."Pump A".size;
       "Pump & Flowrate".pumpA_edited := FALSE;
   END_IF;
   IF "Pump & Flowrate".record_size AND "Pump & Flowrate".pumpB_edited THEN
       "Pump & Flowrate".PumpsizeB_original := "Pump & Flowrate"."Pump B".size;
       "Pump & Flowrate".pumpB_edited := FALSE;
   END_IF;
   IF "Pump & Flowrate".record_size AND NOT "Pump & Flowrate".pumpA_edited AND NOT "Pump & Flowrate".pumpB_edited THEN
       "Pump & Flowrate".record_size := FALSE;
   END_IF;
END_REGION

REGION Network 3
   RUNG wire#powerrail
      "FB0-MR_Quantity Control_1_DB"(RatioCheckMode := "Function Ratio check".input.Mode, AcceptValue := "Function Ratio check".Control.AcceptValue, "Mixing Ratio 100:B" := "Mixing ratio"."Mixing ratio according to density", "Qty A set" := "Function Ratio check".PumpCaliberationControls.CurrentSet_A, "Qty B set" := "Function Ratio check".PumpCaliberationControls.CurrentSet_B, "Pump size A" := "Pump & Flowrate"."Pump A".size, "Pump size B" := "Pump & Flowrate"."Pump B".size, RatioCheckStarted := "Function Ratio check".Control."metering running", DeleteCalibrationA := "Function Ratio check".PumpCaliberationPara."Delete Calibration_A", DeleteCalibrationB := "Function Ratio check".PumpCaliberationPara."Delete Calibration_B", "Qty real A" := "Function Ratio check".PumpCaliberationControls.CurrentActual_A, "Qty real B" := "Function Ratio check".PumpCaliberationControls.CurrentActual_B, "Max. Mixed quantity" =>, "Pump Capacity A cc/rev" =>, "Pump capacity B cc/rev" =>, "cc/rev A" =>, "cc/rev B" =>, "pump adj. ratio A" =>, "pump adj. ratio B" =>, "Total Deviation A" => "Function Ratio check".PumpCaliberationPara.TotalDeviation_A, "Total Deviation B" => "Function Ratio check".PumpCaliberationPara.TotalDeviation_B, "Current Deviation A" => "Function Ratio check".PumpCaliberationPara.CurrentDeviation_A, "Current Deviation B" => "Function Ratio check".PumpCaliberationPara.CurrrentDeviation_B, AllowedMaxAQtyOn2kMetering =>, AllowedMaxBQtyOn2kMetering_1 =>)
   END_RUNG
   // the same network as SCL:
   "FB0-MR_Quantity Control_1_DB"(RatioCheckMode := "Function Ratio check".input.Mode,   // "FB0-MR_Quantity Control_1"
                           AcceptValue := "Function Ratio check".Control.AcceptValue,
                           "Mixing Ratio 100:B" := "Mixing ratio"."Mixing ratio according to density",
                           "Qty A set" := "Function Ratio check".PumpCaliberationControls.CurrentSet_A,
                           "Qty B set" := "Function Ratio check".PumpCaliberationControls.CurrentSet_B,
                           "Pump size A" := "Pump & Flowrate"."Pump A".size,
                           "Pump size B" := "Pump & Flowrate"."Pump B".size,
                           RatioCheckStarted := "Function Ratio check".Control."metering running",
                           DeleteCalibrationA := "Function Ratio check".PumpCaliberationPara."Delete Calibration_A",
                           DeleteCalibrationB := "Function Ratio check".PumpCaliberationPara."Delete Calibration_B",
                           "Qty real A" := "Function Ratio check".PumpCaliberationControls.CurrentActual_A,
                           "Qty real B" := "Function Ratio check".PumpCaliberationControls.CurrentActual_B,
                           "Total Deviation A" => "Function Ratio check".PumpCaliberationPara.TotalDeviation_A,
                           "Total Deviation B" => "Function Ratio check".PumpCaliberationPara.TotalDeviation_B,
                           "Current Deviation A" => "Function Ratio check".PumpCaliberationPara.CurrentDeviation_A,
                           "Current Deviation B" => "Function Ratio check".PumpCaliberationPara.CurrrentDeviation_B);
END_REGION
END_FUNCTION

FUNCTION_BLOCK "FB0-MR_Quantity Control_1"   // FB13, LAD
{ S7_Optimized_Access := 'TRUE' }
VERSION : 0.1
// stored: AutoNumber false, IsIECCheckEnabled false, IsRetainMemResEnabled false, MemoryReserve 100, SetENOAutomatically false, UDAEnableTagReadback false
   VAR_INPUT
      RatioCheckMode : Int;
      AcceptValue : Bool;
      "Mixing Ratio 100:B" : Real;
      "Qty A set" : Real;
      "Qty B set" : Real;
      "Pump size A" : Real;
      "Pump size B" : Real;
      RatioCheckStarted : Bool;
      DeleteCalibrationA : Bool;
      DeleteCalibrationB : Bool;
   END_VAR
   VAR_OUTPUT
      "Max. Mixed quantity" : Real;
      "Pump Capacity A cc/rev" : Real;
      "Pump capacity B cc/rev" : Real;
      "cc/rev A" : Real;
      "cc/rev B" : Real;
      "pump adj. ratio A" : Real;
      "pump adj. ratio B" : Real;
      "Total Deviation A" : Real;
      "Total Deviation B" : Real;
      "Current Deviation A" : Real;
      "Current Deviation B" : Real;
      AllowedMaxAQtyOn2kMetering : Real;
      AllowedMaxBQtyOn2kMetering_1 : Real;
   END_VAR
   VAR_IN_OUT
      "Qty real A" : Real;
      "Qty real B" : Real;
   END_VAR
   VAR RETAIN
      "Last_Cc/rev_A" : Real;
      "Last_Cc/rev_B" : Real;
   END_VAR
   VAR
      "A_Qty/rev_Theor" : Real;
      "B_Qty/rev_Theor" : Real;
      A_Calc_Ref_rev : Real;
      B_Calc_Ref_rev : Real;
      A_Total_Deviation : Real;
      B_Total_Deviation : Real;
   END_VAR
   VAR RETAIN
      B_Current_Deviation : Real;
      A_Current_Deviation : Real;
      "CC/rev actual A" : Real;
      "CC/rev actual B" : Real;
   END_VAR
   VAR
      "A_cc/revStatic_Found" : Real;
      "B_cc/revStatic_Found" : Real;
      "cc/rev calc A" : Real;
      "cc/rev calc B" : Real;
      "Maximum capacity Pump A" : Real;
      "Maximum capacity Pump B" : Real;
      "Individual quantity A MR" : Real;
      "Individual quantity B1 MR" : Real;
      "Individual quantity B MR" : Real;
      "capacity difference" : Real;
      "Ratio margin" : Real;
      "Ratio/100" : Real;
      "Pump cc/rev A" : Real;
      "pump cc/rev B" : Real;
      "A Quantity Compensated" : Real;
      "Quantity A Per ratio" : Real;
      Temp_1 : Bool;
      Last_DeviationA : Real;
      Last_DeviationB : Real;
   END_VAR
   VAR_TEMP   // added for the SCL form of the ladder/FBD networks
      _w1 : Bool;
   END_VAR
BEGIN

REGION Network 1
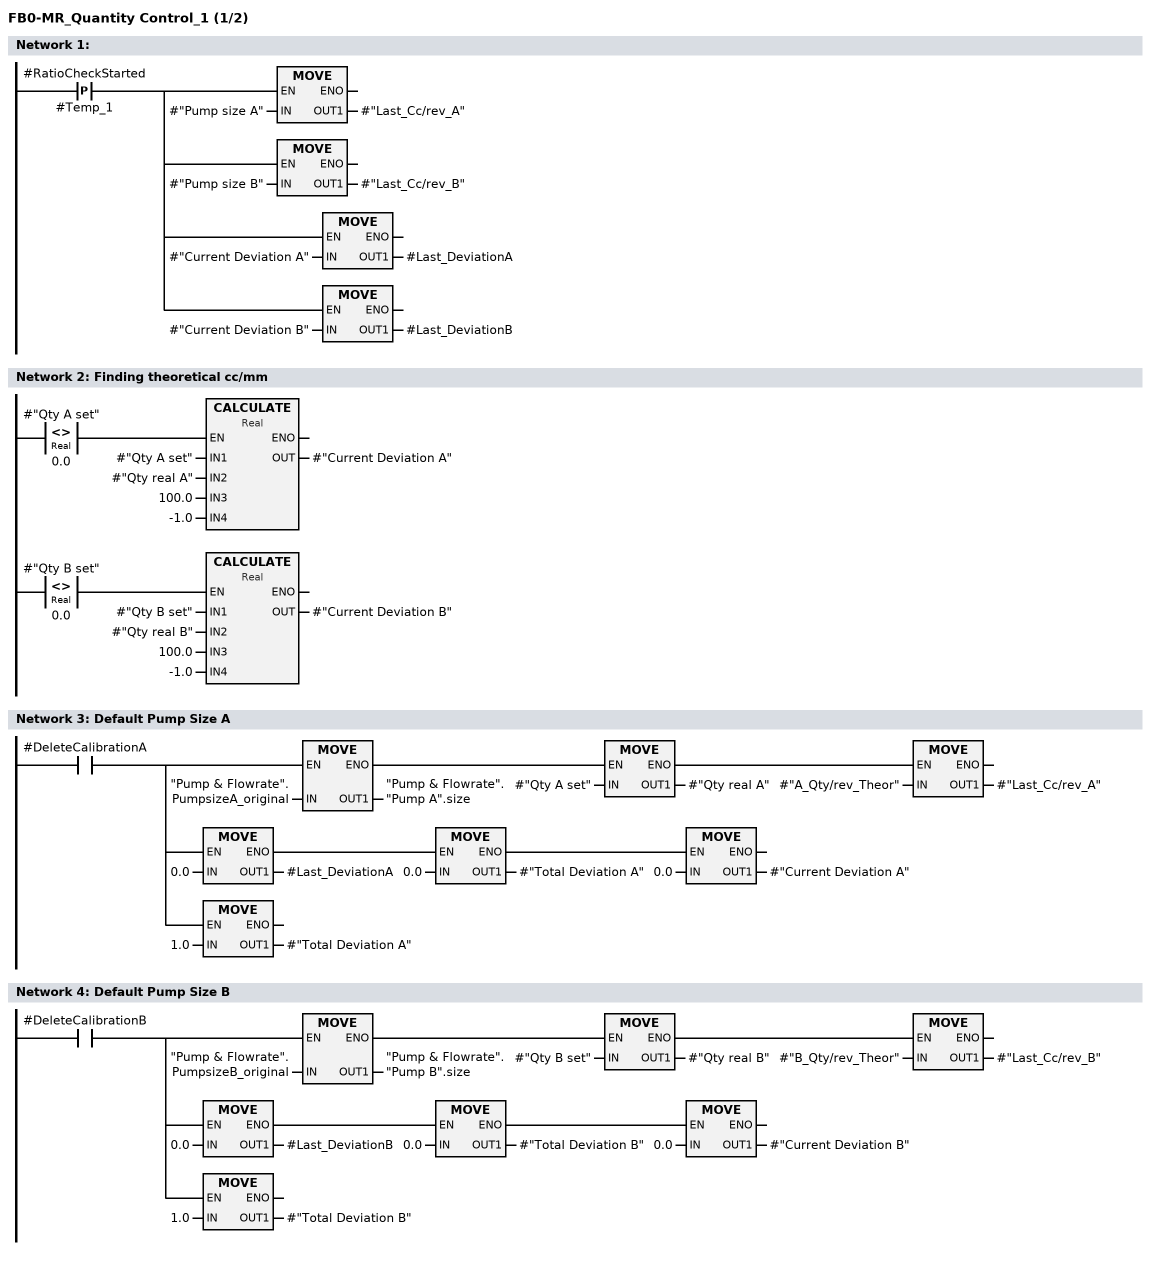
   RUNG wire#powerrail
      P_Contact(operand := #RatioCheckStarted, bit := #Temp_1)
      wire#w1
      Move(in := #"Pump size A", out1 => #"Last_Cc/rev_A")
   END_RUNG
   RUNG wire#w1
      Move(in := #"Pump size B", out1 => #"Last_Cc/rev_B")
   END_RUNG
   RUNG wire#w1
      Move(in := #"Current Deviation A", out1 => #Last_DeviationA)
   END_RUNG
   RUNG wire#w1
      Move(in := #"Current Deviation B", out1 => #Last_DeviationB)
   END_RUNG
   // the same network as SCL:
   #_w1 := #RatioCheckStarted AND NOT #Temp_1;   // rising edge of #RatioCheckStarted
   #Temp_1 := #RatioCheckStarted;
   IF #_w1 THEN
       #"Last_Cc/rev_A" := #"Pump size A";
       #"Last_Cc/rev_B" := #"Pump size B";
       #Last_DeviationA := #"Current Deviation A";
       #Last_DeviationB := #"Current Deviation B";
   END_IF;
END_REGION

REGION Network 2: Finding theoretical cc/mm
   RUNG wire#powerrail
      { S7_Templates := "SrcType := Real" } NE_Contact(in1 := #"Qty A set", in2 := 0.0)
      { S7_Templates := "SrcType := Real"; S7_Expression := "((IN1-IN2)/(IN1/IN3))*(IN4)" } Calculate(in1 := #"Qty A set", in2 := #"Qty real A", in3 := 100.0, in4 := -1.0, out => #"Current Deviation A")
   END_RUNG
   RUNG wire#powerrail
      { S7_Templates := "SrcType := Real" } NE_Contact(in1 := #"Qty B set", in2 := 0.0)
      { S7_Templates := "SrcType := Real"; S7_Expression := "(IN1-IN2)/(IN1/IN3)*(IN4)" } Calculate(in1 := #"Qty B set", in2 := #"Qty real B", in3 := 100.0, in4 := -1.0, out => #"Current Deviation B")
   END_RUNG
   // the same network as SCL:
   IF #"Qty A set" <> 0.0 THEN
       #"Current Deviation A" := ((#"Qty A set"-#"Qty real A")/(#"Qty A set"/100.0))*((-1.0));
   END_IF;
   IF #"Qty B set" <> 0.0 THEN
       #"Current Deviation B" := (#"Qty B set"-#"Qty real B")/(#"Qty B set"/100.0)*((-1.0));
   END_IF;
END_REGION

REGION Network 3: Default Pump Size A
   IF #DeleteCalibrationA THEN
       "Pump & Flowrate"."Pump A".size := "Pump & Flowrate".PumpsizeA_original;
       #"Qty real A" := #"Qty A set";
       #"Last_Cc/rev_A" := #"A_Qty/rev_Theor";
       #Last_DeviationA := 0.0;
       #"Total Deviation A" := 0.0;
       #"Current Deviation A" := 0.0;
       #"Total Deviation A" := 1.0;
   END_IF;
END_REGION

REGION Network 4: Default Pump Size B
   IF #DeleteCalibrationB THEN
       "Pump & Flowrate"."Pump B".size := "Pump & Flowrate".PumpsizeB_original;
       #"Qty real B" := #"Qty B set";
       #"Last_Cc/rev_B" := #"B_Qty/rev_Theor";
       #Last_DeviationB := 0.0;
       #"Total Deviation B" := 0.0;
       #"Current Deviation B" := 0.0;
       #"Total Deviation B" := 1.0;
   END_IF;
END_REGION

REGION Network 5
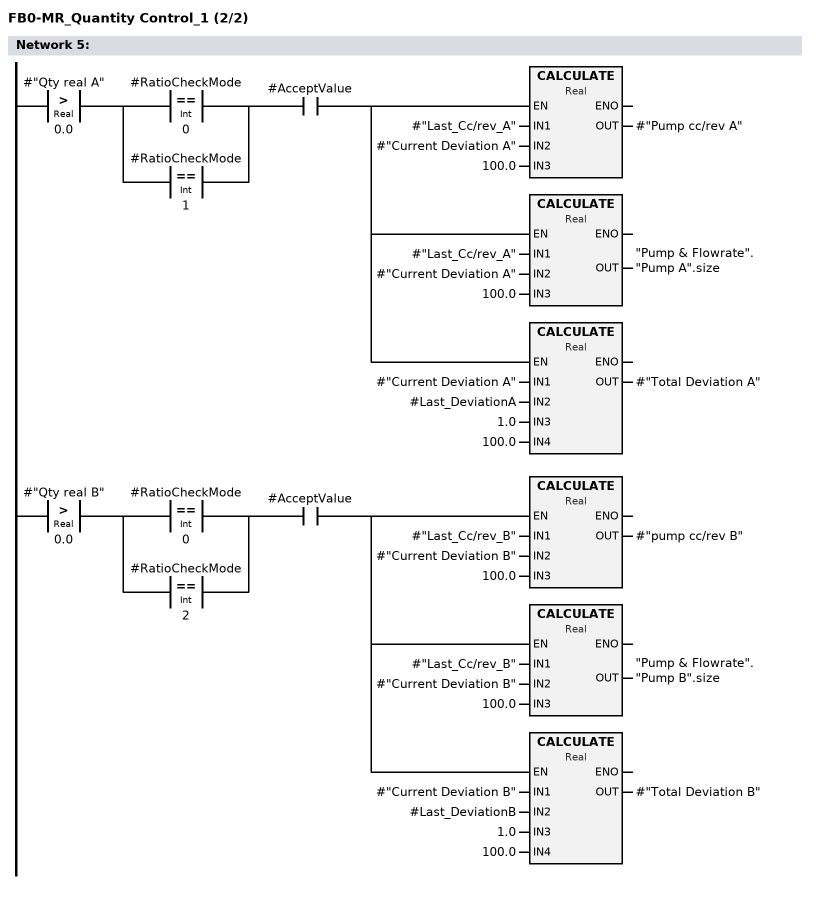
   IF (#"Qty real A" > 0.0) AND ((#RatioCheckMode = 0) OR (#RatioCheckMode = 1)) AND #AcceptValue THEN
       #"Pump cc/rev A" := #"Last_Cc/rev_A"+(#"Last_Cc/rev_A"*(#"Current Deviation A"/100.0));
       "Pump & Flowrate"."Pump A".size := #"Last_Cc/rev_A"+(#"Last_Cc/rev_A"*(#"Current Deviation A"/100.0));
       #"Total Deviation A" := 1.0-((#"Current Deviation A"+#Last_DeviationA)/100.0);
   END_IF;
   IF (#"Qty real B" > 0.0) AND ((#RatioCheckMode = 0) OR (#RatioCheckMode = 2)) AND #AcceptValue THEN
       #"pump cc/rev B" := #"Last_Cc/rev_B"+(#"Last_Cc/rev_B"*(#"Current Deviation B"/100.0));
       "Pump & Flowrate"."Pump B".size := #"Last_Cc/rev_B"+(#"Last_Cc/rev_B"*(#"Current Deviation B"/100.0));
       #"Total Deviation B" := 1.0-((#"Current Deviation B"+#Last_DeviationB)/100.0);
   END_IF;
END_REGION
END_FUNCTION_BLOCK

FUNCTION "Heater" : Void   // FC34, LAD
{ S7_Optimized_Access := 'TRUE' }
VERSION : 0.1
// stored: AutoNumber true, IsIECCheckEnabled false, SetENOAutomatically true, UDAEnableTagReadback false
BEGIN

REGION Network 1 (SCL): Show Heater button if any of the heaters active
   IF "Heater settings"."heater EN 1" OR "Heater settings"."heater EN 2" OR
       "Heater settings"."heater EN 3" OR"Heater settings"."heater EN 4" THEN
       "Heatercontrol"."Show heater Button" := TRUE;
   ELSE
       "Heatercontrol"."Show heater Button" := false;
   END_IF;

   IF "Heatercontrol"."Show heater Button" = false THEN
       "Heatercontrol"."heater ON HMI" := false;
   END_IF;
END_REGION

REGION Network 2 (SCL): Actual temperature of RTD Sensor
   // heaters from 1 to 8 IW144 to IW158 //

   IF "heater1" >= 32767 THEN
       "heater status".temperature.heater1 := 0;
   ELSE
       "heater status".temperature.heater1 := "heater1" / 10;
   END_IF;
   IF "heater2" >= 32767 THEN
       "heater status".temperature.heater2 := 0;
   ELSE
       "heater status".temperature.heater2 := "heater2" / 10;
   END_IF;
   IF "heater3" >= 32767 THEN
       "heater status".temperature.heater3 := 0;
   ELSE
       "heater status".temperature.heater3 := "heater3" / 10;
   END_IF;
   IF "heater4" >= 32767 THEN
       "heater status".temperature.heater4 := 0;
   ELSE
       "heater status".temperature.heater4 := "heater4" / 10;
   END_IF;
END_REGION

REGION Network 3 (SCL): Pt-100 Sensor Connection Okay
   // heaters from 1 to 8 IW144 to IW158 //
   "heater status"."p100 connection okay".heater1 := ("heater1" < 32727);
   "heater status"."p100 connection okay".heater2 := ("heater2" < 32727);
   "heater status"."p100 connection okay".heater3 := ("heater3" < 32727);
   "heater status"."p100 connection okay".heater4 := ("heater4" < 32727);
END_REGION

REGION Network 4 (SCL): alarm
   "Alarm_DB".input.alarm[3] := NOT ("heater status"."p100 connection okay".heater1) AND "Heater settings"."heater EN 1"; //A12-Heater1 sensor fault
   "Alarm_DB".input.alarm[4] := NOT ("heater status"."p100 connection okay".heater2) AND "Heater settings"."heater EN 2";  //A13-Heater1 sensor fault
   "Alarm_DB".input.alarm[5] := NOT ("heater status"."p100 connection okay".heater3) AND "Heater settings"."heater EN 3"; //A14-Heater3 sensor fault
   "Alarm_DB".input.alarm[6] := NOT ("heater status"."p100 connection okay".heater4) AND "Heater settings"."heater EN 4";  //A15-Heater4 sensor fault


   "Alarm_DB".input.alarm[28] := "heater status"."Limit Over temperature".heater1; //"A21- Heater 1overtemperature"
   "Alarm_DB".input.alarm[29] := "heater status"."Limit Over temperature".heater2; //"A22- Heater2 overtemperature"
   "Alarm_DB".input.alarm[30] := "heater status"."Limit Over temperature".heater3; //"A23- Heater3 overtemperature"
   "Alarm_DB".input.alarm[31] := "heater status"."Limit Over temperature".heater4; //"A24- Heater4 overtemperature"

   "Alarm_DB".input.alarm[24] := ("heater status"."Dispensing Stop under temperature heater"[1] AND "Heater settings"."heater EN 1") OR "heater status"."Limit under temperature".heater1;
   "Alarm_DB".input.alarm[25] := ("heater status"."Dispensing Stop under temperature heater"[2] AND "Heater settings"."heater EN 2") OR "heater status"."Limit under temperature".heater2;
   "Alarm_DB".input.alarm[26] := ("heater status"."Dispensing Stop under temperature heater"[3] AND "Heater settings"."heater EN 3") OR "heater status"."Limit under temperature".heater3;
   "Alarm_DB".input.alarm[27] := ("heater status"."Dispensing Stop under temperature heater"[4] AND "Heater settings"."heater EN 4") OR "heater status"."Limit under temperature".heater4;
END_REGION

REGION Network 5: heater 1- Vessel heating sleeve A component
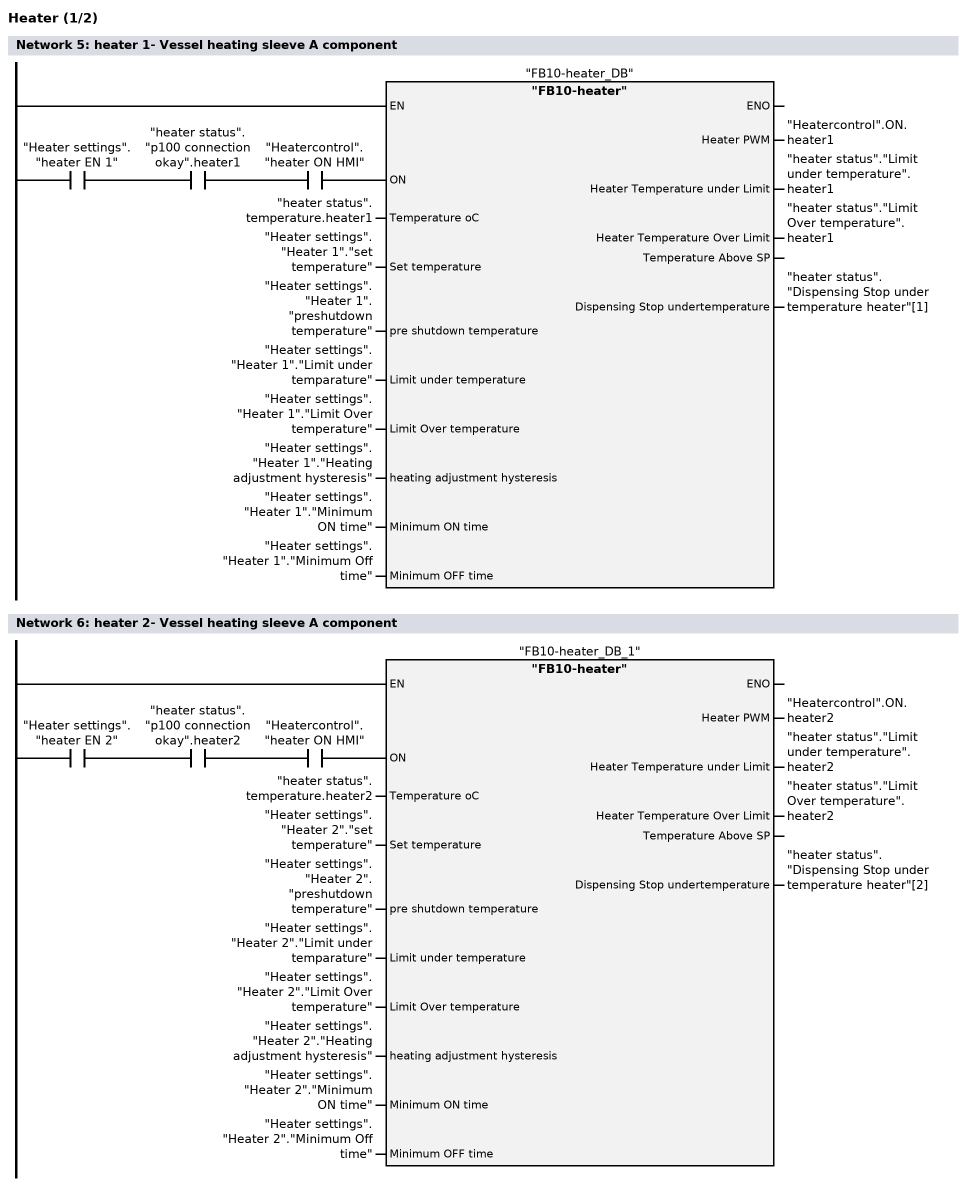
   RUNG wire#powerrail
      "FB10-heater_DB"(ON := wire#w1, "Temperature oC" := "heater status".temperature.heater1, "Set temperature" := "Heater settings"."Heater 1"."set temperature", "pre shutdown temperature" := "Heater settings"."Heater 1"."preshutdown temperature", "Limit under temperature" := "Heater settings"."Heater 1"."Limit under temparature", "Limit Over temperature" := "Heater settings"."Heater 1"."Limit Over temperature", "heating adjustment hysteresis" := "Heater settings"."Heater 1"."Heating adjustment hysteresis", "Minimum ON time" := "Heater settings"."Heater 1"."Minimum ON time", "Minimum OFF time" := "Heater settings"."Heater 1"."Minimum Off time", "Heater PWM" => "Heatercontrol".ON.heater1, "Heater Temperature under Limit" => "heater status"."Limit under temperature".heater1, "Heater Temperature Over Limit" => "heater status"."Limit Over temperature".heater1, "Temperature Above SP" =>, "Dispensing Stop undertemperature" => "heater status"."Dispensing Stop under temperature heater"[1])
   END_RUNG
   RUNG wire#powerrail
      Contact( "Heater settings"."heater EN 1" )
      Contact( "heater status"."p100 connection okay".heater1 )
      Contact( "Heatercontrol"."heater ON HMI" )
   END_RUNG wire#w1
   // the same network as SCL:
   "FB10-heater_DB"(ON := "Heater settings"."heater EN 1" AND "heater status"."p100 connection okay".heater1 AND "Heatercontrol"."heater ON HMI",   // "FB10-heater"
                    "Temperature oC" := "heater status".temperature.heater1,
                    "Set temperature" := "Heater settings"."Heater 1"."set temperature",
                    "pre shutdown temperature" := "Heater settings"."Heater 1"."preshutdown temperature",
                    "Limit under temperature" := "Heater settings"."Heater 1"."Limit under temparature",
                    "Limit Over temperature" := "Heater settings"."Heater 1"."Limit Over temperature",
                    "heating adjustment hysteresis" := "Heater settings"."Heater 1"."Heating adjustment hysteresis",
                    "Minimum ON time" := "Heater settings"."Heater 1"."Minimum ON time",
                    "Minimum OFF time" := "Heater settings"."Heater 1"."Minimum Off time",
                    "Heater PWM" => "Heatercontrol".ON.heater1,
                    "Heater Temperature under Limit" => "heater status"."Limit under temperature".heater1,
                    "Heater Temperature Over Limit" => "heater status"."Limit Over temperature".heater1,
                    "Dispensing Stop undertemperature" => "heater status"."Dispensing Stop under temperature heater"[1]);
END_REGION

REGION Network 6: heater 2- Vessel heating sleeve A component
   RUNG wire#powerrail
      "FB10-heater_DB_1"(ON := wire#w1, "Temperature oC" := "heater status".temperature.heater2, "Set temperature" := "Heater settings"."Heater 2"."set temperature", "pre shutdown temperature" := "Heater settings"."Heater 2"."preshutdown temperature", "Limit under temperature" := "Heater settings"."Heater 2"."Limit under temparature", "Limit Over temperature" := "Heater settings"."Heater 2"."Limit Over temperature", "heating adjustment hysteresis" := "Heater settings"."Heater 2"."Heating adjustment hysteresis", "Minimum ON time" := "Heater settings"."Heater 2"."Minimum ON time", "Minimum OFF time" := "Heater settings"."Heater 2"."Minimum Off time", "Heater PWM" => "Heatercontrol".ON.heater2, "Heater Temperature under Limit" => "heater status"."Limit under temperature".heater2, "Heater Temperature Over Limit" => "heater status"."Limit Over temperature".heater2, "Temperature Above SP" =>, "Dispensing Stop undertemperature" => "heater status"."Dispensing Stop under temperature heater"[2])
   END_RUNG
   RUNG wire#powerrail
      Contact( "Heater settings"."heater EN 2" )
      Contact( "heater status"."p100 connection okay".heater2 )
      Contact( "Heatercontrol"."heater ON HMI" )
   END_RUNG wire#w1
   // the same network as SCL:
   "FB10-heater_DB_1"(ON := "Heater settings"."heater EN 2" AND "heater status"."p100 connection okay".heater2 AND "Heatercontrol"."heater ON HMI",   // "FB10-heater"
                      "Temperature oC" := "heater status".temperature.heater2,
                      "Set temperature" := "Heater settings"."Heater 2"."set temperature",
                      "pre shutdown temperature" := "Heater settings"."Heater 2"."preshutdown temperature",
                      "Limit under temperature" := "Heater settings"."Heater 2"."Limit under temparature",
                      "Limit Over temperature" := "Heater settings"."Heater 2"."Limit Over temperature",
                      "heating adjustment hysteresis" := "Heater settings"."Heater 2"."Heating adjustment hysteresis",
                      "Minimum ON time" := "Heater settings"."Heater 2"."Minimum ON time",
                      "Minimum OFF time" := "Heater settings"."Heater 2"."Minimum Off time",
                      "Heater PWM" => "Heatercontrol".ON.heater2,
                      "Heater Temperature under Limit" => "heater status"."Limit under temperature".heater2,
                      "Heater Temperature Over Limit" => "heater status"."Limit Over temperature".heater2,
                      "Dispensing Stop undertemperature" => "heater status"."Dispensing Stop under temperature heater"[2]);
END_REGION

REGION Network 7: heater 3- Heating sleeve flowmeter A component
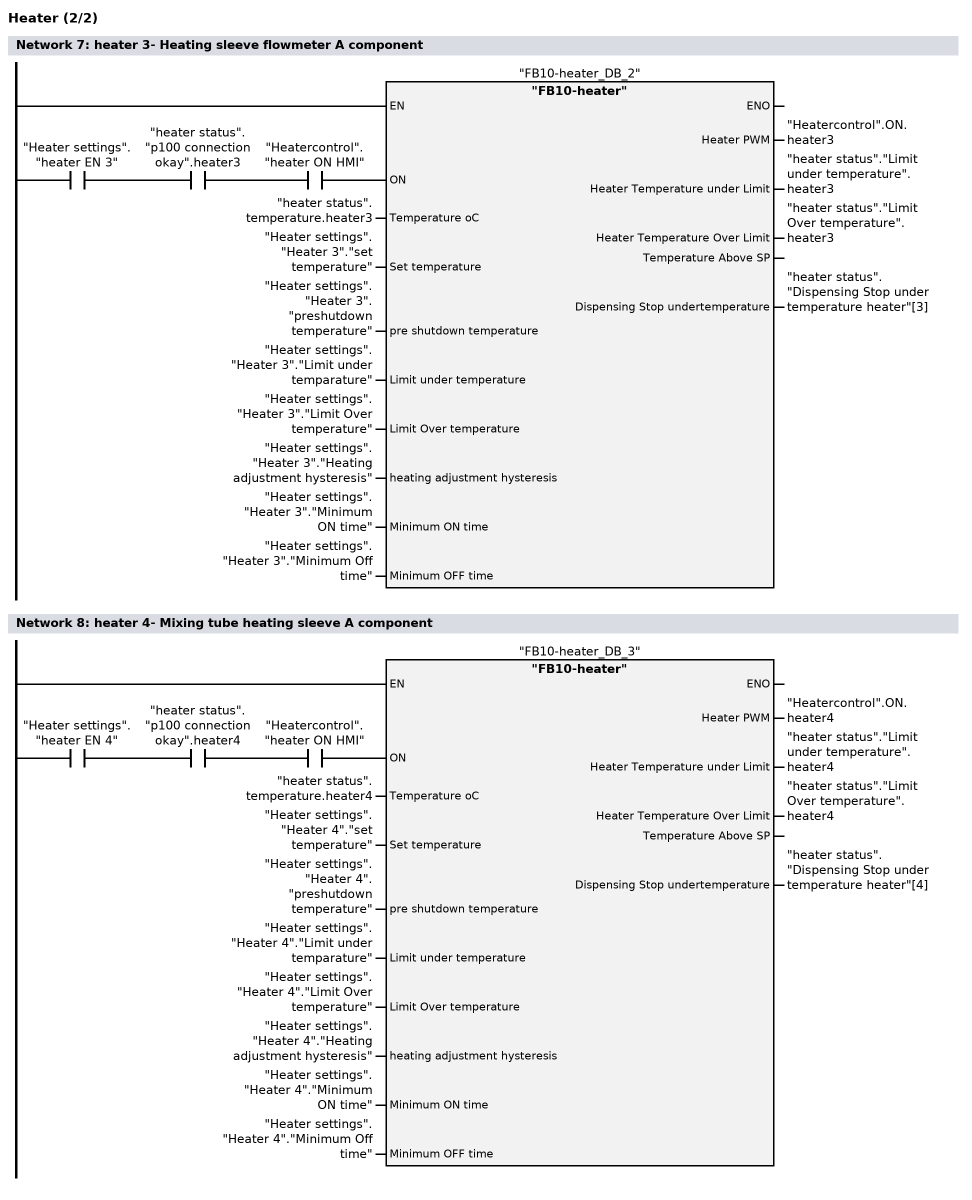
   RUNG wire#powerrail
      "FB10-heater_DB_2"(ON := wire#w1, "Temperature oC" := "heater status".temperature.heater3, "Set temperature" := "Heater settings"."Heater 3"."set temperature", "pre shutdown temperature" := "Heater settings"."Heater 3"."preshutdown temperature", "Limit under temperature" := "Heater settings"."Heater 3"."Limit under temparature", "Limit Over temperature" := "Heater settings"."Heater 3"."Limit Over temperature", "heating adjustment hysteresis" := "Heater settings"."Heater 3"."Heating adjustment hysteresis", "Minimum ON time" := "Heater settings"."Heater 3"."Minimum ON time", "Minimum OFF time" := "Heater settings"."Heater 3"."Minimum Off time", "Heater PWM" => "Heatercontrol".ON.heater3, "Heater Temperature under Limit" => "heater status"."Limit under temperature".heater3, "Heater Temperature Over Limit" => "heater status"."Limit Over temperature".heater3, "Temperature Above SP" =>, "Dispensing Stop undertemperature" => "heater status"."Dispensing Stop under temperature heater"[3])
   END_RUNG
   RUNG wire#powerrail
      Contact( "Heater settings"."heater EN 3" )
      Contact( "heater status"."p100 connection okay".heater3 )
      Contact( "Heatercontrol"."heater ON HMI" )
   END_RUNG wire#w1
   // the same network as SCL:
   "FB10-heater_DB_2"(ON := "Heater settings"."heater EN 3" AND "heater status"."p100 connection okay".heater3 AND "Heatercontrol"."heater ON HMI",   // "FB10-heater"
                      "Temperature oC" := "heater status".temperature.heater3,
                      "Set temperature" := "Heater settings"."Heater 3"."set temperature",
                      "pre shutdown temperature" := "Heater settings"."Heater 3"."preshutdown temperature",
                      "Limit under temperature" := "Heater settings"."Heater 3"."Limit under temparature",
                      "Limit Over temperature" := "Heater settings"."Heater 3"."Limit Over temperature",
                      "heating adjustment hysteresis" := "Heater settings"."Heater 3"."Heating adjustment hysteresis",
                      "Minimum ON time" := "Heater settings"."Heater 3"."Minimum ON time",
                      "Minimum OFF time" := "Heater settings"."Heater 3"."Minimum Off time",
                      "Heater PWM" => "Heatercontrol".ON.heater3,
                      "Heater Temperature under Limit" => "heater status"."Limit under temperature".heater3,
                      "Heater Temperature Over Limit" => "heater status"."Limit Over temperature".heater3,
                      "Dispensing Stop undertemperature" => "heater status"."Dispensing Stop under temperature heater"[3]);
END_REGION

REGION Network 8: heater 4- Mixing tube heating sleeve A component
   RUNG wire#powerrail
      "FB10-heater_DB_3"(ON := wire#w1, "Temperature oC" := "heater status".temperature.heater4, "Set temperature" := "Heater settings"."Heater 4"."set temperature", "pre shutdown temperature" := "Heater settings"."Heater 4"."preshutdown temperature", "Limit under temperature" := "Heater settings"."Heater 4"."Limit under temparature", "Limit Over temperature" := "Heater settings"."Heater 4"."Limit Over temperature", "heating adjustment hysteresis" := "Heater settings"."Heater 4"."Heating adjustment hysteresis", "Minimum ON time" := "Heater settings"."Heater 4"."Minimum ON time", "Minimum OFF time" := "Heater settings"."Heater 4"."Minimum Off time", "Heater PWM" => "Heatercontrol".ON.heater4, "Heater Temperature under Limit" => "heater status"."Limit under temperature".heater4, "Heater Temperature Over Limit" => "heater status"."Limit Over temperature".heater4, "Temperature Above SP" =>, "Dispensing Stop undertemperature" => "heater status"."Dispensing Stop under temperature heater"[4])
   END_RUNG
   RUNG wire#powerrail
      Contact( "Heater settings"."heater EN 4" )
      Contact( "heater status"."p100 connection okay".heater4 )
      Contact( "Heatercontrol"."heater ON HMI" )
   END_RUNG wire#w1
   // the same network as SCL:
   "FB10-heater_DB_3"(ON := "Heater settings"."heater EN 4" AND "heater status"."p100 connection okay".heater4 AND "Heatercontrol"."heater ON HMI",   // "FB10-heater"
                      "Temperature oC" := "heater status".temperature.heater4,
                      "Set temperature" := "Heater settings"."Heater 4"."set temperature",
                      "pre shutdown temperature" := "Heater settings"."Heater 4"."preshutdown temperature",
                      "Limit under temperature" := "Heater settings"."Heater 4"."Limit under temparature",
                      "Limit Over temperature" := "Heater settings"."Heater 4"."Limit Over temperature",
                      "heating adjustment hysteresis" := "Heater settings"."Heater 4"."Heating adjustment hysteresis",
                      "Minimum ON time" := "Heater settings"."Heater 4"."Minimum ON time",
                      "Minimum OFF time" := "Heater settings"."Heater 4"."Minimum Off time",
                      "Heater PWM" => "Heatercontrol".ON.heater4,
                      "Heater Temperature under Limit" => "heater status"."Limit under temperature".heater4,
                      "Heater Temperature Over Limit" => "heater status"."Limit Over temperature".heater4,
                      "Dispensing Stop undertemperature" => "heater status"."Dispensing Stop under temperature heater"[4]);
END_REGION

REGION Network 9 (SCL): Stop Dispensing when Temperature Not Okay During under temperature Without making heater ON
   IF ("heater status"."Dispensing Stop under temperature heater"[1] AND "Heater settings"."heater EN 1") OR
       ("heater status"."Dispensing Stop under temperature heater"[2] AND "Heater settings"."heater EN 2") OR
       ("heater status"."Dispensing Stop under temperature heater"[3] AND "Heater settings"."heater EN 3") OR
       ("heater status"."Dispensing Stop under temperature heater"[4] AND "Heater settings"."heater EN 4")OR
       "heater status".heater_nok
   THEN
     "heater status"."Critical Fault Stop Dispense Temperature NOK" := 1;
   ELSE
     "heater status"."Critical Fault Stop Dispense Temperature NOK" := 0;
   END_IF;
END_REGION
END_FUNCTION

FUNCTION_BLOCK "FB10-heater"   // FB12, LAD
{ S7_Optimized_Access := 'TRUE' }
VERSION : 0.1
// stored: AutoNumber true, IsIECCheckEnabled false, IsRetainMemResEnabled false, MemoryReserve 100, SetENOAutomatically false, UDAEnableTagReadback false
   VAR_INPUT
      ON : Bool;
      "Temperature oC" : Real;
      "Set temperature" : Real;
      "pre shutdown temperature" : Real;
      "Limit under temperature" : Real;
      "Limit Over temperature" : Real;
      "heating adjustment hysteresis" : Real;
      "Minimum ON time" : Real;
      "Minimum OFF time" : Real;
   END_VAR
   VAR_OUTPUT
      "Heater PWM" : Bool;
      "Heater Temperature under Limit" : Bool;
      "Heater Temperature Over Limit" : Bool;
      "Temperature Above SP" { ExternalAccessible := 'False'; ExternalVisible := 'False'; ExternalWritable := 'False'} : Bool;
      "Dispensing Stop undertemperature" { ExternalAccessible := 'False'; ExternalVisible := 'False'; ExternalWritable := 'False'} : Bool;
   END_VAR
   VAR
      "set temperature after hysteresis" : Real;
      "On time in msec" : DInt;
      "off time in msec" : DInt;
      "On timer triggered" : Bool;
      "off time triggered" : Bool;
      IEC_Timer_0_Instance { S7_SetPoint := 'True'} : TON_TIME;
      IEC_Timer_0_Instance_1 { S7_SetPoint := 'True'} : TON_TIME;
   END_VAR
   VAR_TEMP   // added for the SCL form of the ladder/FBD networks
      _w1 : Bool;
   END_VAR
BEGIN

REGION Network 1: On/off timer in sec
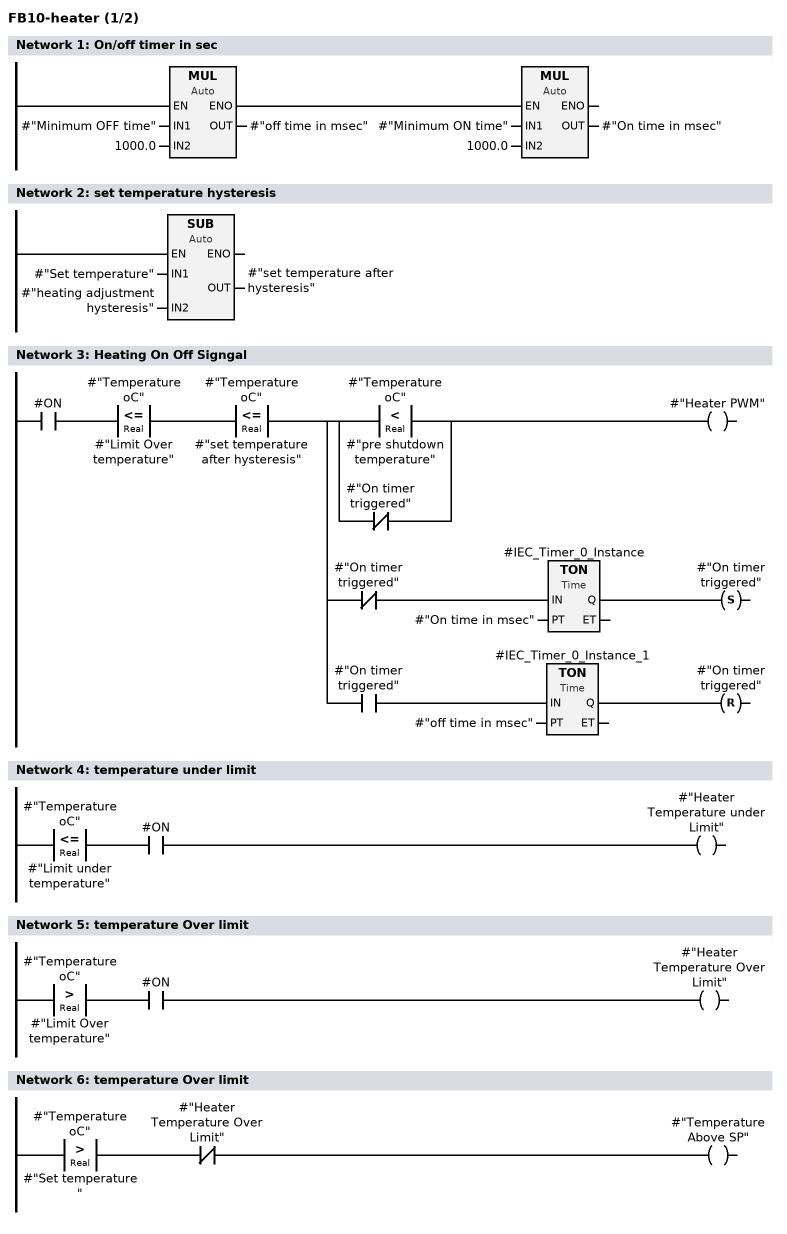
   RUNG wire#powerrail
      Mul(in1 := #"Minimum OFF time", in2 := 1000.0, out => #"off time in msec")
      Mul(in1 := #"Minimum ON time", in2 := 1000.0, out => #"On time in msec")
   END_RUNG
   // the same network as SCL:
   #"off time in msec" := #"Minimum OFF time" * 1000.0;
   #"On time in msec" := #"Minimum ON time" * 1000.0;
END_REGION

REGION Network 2: set temperature hysteresis
   RUNG wire#powerrail
      Sub(in1 := #"Set temperature", in2 := #"heating adjustment hysteresis", out => #"set temperature after hysteresis")
   END_RUNG
   // the same network as SCL:
   #"set temperature after hysteresis" := #"Set temperature" - #"heating adjustment hysteresis";
END_REGION

REGION Network 3: Heating On Off Signgal
   RUNG wire#powerrail
      Contact( #ON )
      { S7_Templates := "SrcType := Real" } LE_Contact(in1 := #"Temperature oC", in2 := #"Limit Over temperature")
      { S7_Templates := "SrcType := Real" } LE_Contact(in1 := #"Temperature oC", in2 := #"set temperature after hysteresis")
      wire#w1
      { S7_Templates := "SrcType := Real" } LT_Contact(in1 := #"Temperature oC", in2 := #"pre shutdown temperature")
      wire#w2
      Coil( #"Heater PWM" )
   END_RUNG
   RUNG wire#w1
      I_Contact( #"On timer triggered" )
   END_RUNG wire#w2
   RUNG wire#w1
      I_Contact( #"On timer triggered" )
      { S7_Templates := "time_type := Time" } #IEC_Timer_0_Instance.TON(pt := #"On time in msec", et =>)
      S_Coil( #"On timer triggered" )
   END_RUNG
   RUNG wire#w1
      Contact( #"On timer triggered" )
      { S7_Templates := "time_type := Time" } #IEC_Timer_0_Instance_1.TON(pt := #"off time in msec", et =>)
      R_Coil( #"On timer triggered" )
   END_RUNG
   // the same network as SCL:
   #_w1 := #ON AND (#"Temperature oC" <= #"Limit Over temperature") AND (#"Temperature oC" <= #"set temperature after hysteresis");
   #"Heater PWM" := #_w1 AND ((#"Temperature oC" < #"pre shutdown temperature") OR NOT #"On timer triggered");
   #IEC_Timer_0_Instance(IN := #_w1 AND NOT #"On timer triggered", PT := #"On time in msec");   // TON
   IF #IEC_Timer_0_Instance.Q THEN #"On timer triggered" := TRUE; END_IF;
   #IEC_Timer_0_Instance_1(IN := #_w1 AND #"On timer triggered", PT := #"off time in msec");   // TON
   IF #IEC_Timer_0_Instance_1.Q THEN #"On timer triggered" := FALSE; END_IF;
END_REGION

REGION Network 4: temperature under limit
   RUNG wire#powerrail
      { S7_Templates := "SrcType := Real" } LE_Contact(in1 := #"Temperature oC", in2 := #"Limit under temperature")
      Contact( #ON )
      Coil( #"Heater Temperature under Limit" )
   END_RUNG
   // the same network as SCL:
   #"Heater Temperature under Limit" := (#"Temperature oC" <= #"Limit under temperature") AND #ON;
END_REGION

REGION Network 5: temperature Over limit
   RUNG wire#powerrail
      { S7_Templates := "SrcType := Real" } GT_Contact(in1 := #"Temperature oC", in2 := #"Limit Over temperature")
      Contact( #ON )
      Coil( #"Heater Temperature Over Limit" )
   END_RUNG
   // the same network as SCL:
   #"Heater Temperature Over Limit" := (#"Temperature oC" > #"Limit Over temperature") AND #ON;
END_REGION

REGION Network 6: temperature Over limit
   RUNG wire#powerrail
      { S7_Templates := "SrcType := Real" } GT_Contact(in1 := #"Temperature oC", in2 := #"Set temperature")
      I_Contact( #"Heater Temperature Over Limit" )
      Coil( #"Temperature Above SP" )
   END_RUNG
   // the same network as SCL:
   #"Temperature Above SP" := (#"Temperature oC" > #"Set temperature") AND NOT #"Heater Temperature Over Limit";
END_REGION

REGION Network 7: Temperature Under limit to Stop Dispensing
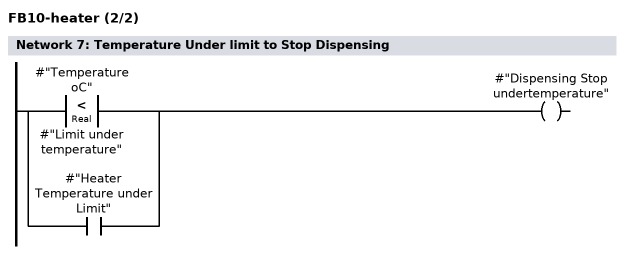
   RUNG wire#powerrail
      { S7_Templates := "SrcType := Real" } LT_Contact(in1 := #"Temperature oC", in2 := #"Limit under temperature")
      wire#w1
      Coil( #"Dispensing Stop undertemperature" )
   END_RUNG
   RUNG wire#powerrail
      Contact( #"Heater Temperature under Limit" )
   END_RUNG wire#w1
   // the same network as SCL:
   #"Dispensing Stop undertemperature" := (#"Temperature oC" < #"Limit under temperature") OR #"Heater Temperature under Limit";
END_REGION
END_FUNCTION_BLOCK

FUNCTION_BLOCK "FB1-MR_Flowrate Control"   // FB1, LAD
{ S7_Optimized_Access := 'TRUE' }
VERSION : 0.1
// stored: AutoNumber true, IsIECCheckEnabled false, IsRetainMemResEnabled false, MemoryReserve 100, SetENOAutomatically false, UDAEnableTagReadback false
   VAR_INPUT
      "Pump size A" : Real;
      "pump size B" : Real;
      "Pump speed A" : Real;
      "pump Speed B" : Real;
      "Mixing Ratio 100:B" : Real;
      "Metering Qty" : Real;
      "Metering Flowrate" : Real;
      "Flowrate Adjustemnt A %" : Real;
      "Flowrate Adjustment B %" : Real;
      "Pump A max Hz" : Real;
      "pump B max Hz" : Real;
   END_VAR
   VAR_OUTPUT
      "Flowrate pump A without adjustment" : Real;
      "Flowrate pump B without adjustment" : Real;
      "Flowrate pump A with adjustment" : Real;
      "Flowrate pump B with adjustment" : Real;
      "Mixed Flowrate" : Real;
      "Pump Capacity A cc/min" : Real;
      "Pump capacity B cc/min" : Real;
      "Pump A frequency" : Real;
      "Pump B frequency" : Real;
      "Metering time" : DInt;
      "Meteringtime in sec" : Int;
   END_VAR
   VAR
      "Maximum Flowrate Pump A" : Real;
      "Maximum Flowrate Pump B" : Real;
      "Pump compensation" : Real;
      "Individual flowrate A MR" : Real;
      "Individual flowrate B1 MR" : Real;
      "Individual flowrate B MR" : Real;
      "Flowrate Ratio difference A" : Real;
      "Flowrate Ratio difference B" : Real;
      "Flowrate Pump A" : Real;
      "Flowrate Pump B" : Real;
      "Flowrate B After Compensation" : Real;
      "Mixed flowrate A+B" : Real;
      "Flowrate to adjust A" : Real;
      "Flowrate to adjust B" : Real;
      "metering time in minutes" : Real;
      "metering time in Sec" : Real;
      "Metering time in msec" : LReal;
      "flowrate to adjust A_1" : Real;
      "flowrate to adjust B_1" : Real;
      "Ratio>100" : Real;
      "amount to reduce in A" : Real;
      "Flowrate difference" : Real;
      "Ratio margin" : Real;
      "Ratio/100" : Real;
      "Flowrate A Per ratio" : Real;
      "A Flowrate Compensated" : Real;
   END_VAR
BEGIN

REGION Network 1: Pump Size and speed multiplication
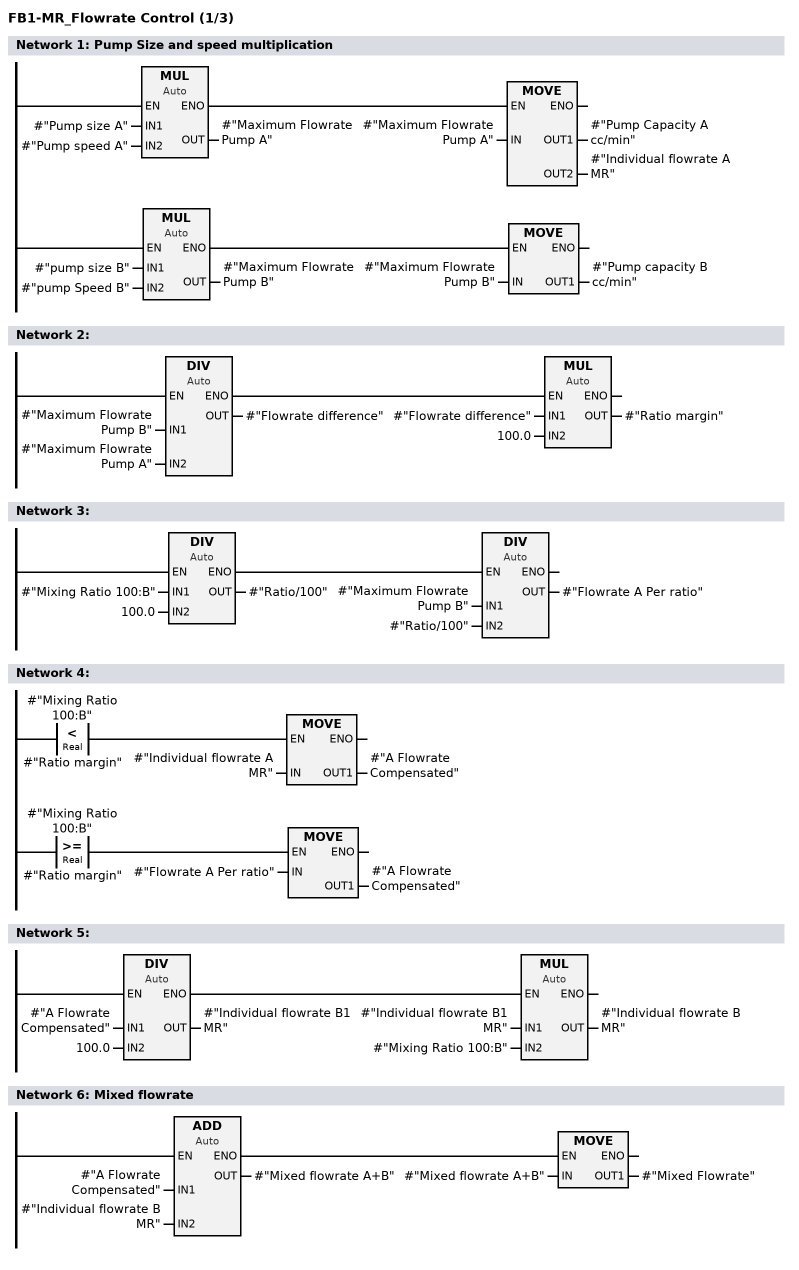
   RUNG wire#powerrail
      Mul(in1 := #"Pump size A", in2 := #"Pump speed A", out => #"Maximum Flowrate Pump A")
      Move(in := #"Maximum Flowrate Pump A", out1 => #"Pump Capacity A cc/min", out2 => #"Individual flowrate A MR")
   END_RUNG
   RUNG wire#powerrail
      Mul(in1 := #"pump size B", in2 := #"pump Speed B", out => #"Maximum Flowrate Pump B")
      Move(in := #"Maximum Flowrate Pump B", out1 => #"Pump capacity B cc/min")
   END_RUNG
   // the same network as SCL:
   #"Maximum Flowrate Pump A" := #"Pump size A" * #"Pump speed A";
   #"Pump Capacity A cc/min" := #"Maximum Flowrate Pump A";
   #"Individual flowrate A MR" := #"Maximum Flowrate Pump A";
   #"Maximum Flowrate Pump B" := #"pump size B" * #"pump Speed B";
   #"Pump capacity B cc/min" := #"Maximum Flowrate Pump B";
END_REGION

REGION Network 2
   RUNG wire#powerrail
      Div(in1 := #"Maximum Flowrate Pump B", in2 := #"Maximum Flowrate Pump A", out => #"Flowrate difference")
      Mul(in1 := #"Flowrate difference", in2 := 100.0, out => #"Ratio margin")
   END_RUNG
   // the same network as SCL:
   #"Flowrate difference" := #"Maximum Flowrate Pump B" / #"Maximum Flowrate Pump A";
   #"Ratio margin" := #"Flowrate difference" * 100.0;
END_REGION

REGION Network 3
   RUNG wire#powerrail
      Div(in1 := #"Mixing Ratio 100:B", in2 := 100.0, out => #"Ratio/100")
      Div(in1 := #"Maximum Flowrate Pump B", in2 := #"Ratio/100", out => #"Flowrate A Per ratio")
   END_RUNG
   // the same network as SCL:
   #"Ratio/100" := #"Mixing Ratio 100:B" / 100.0;
   #"Flowrate A Per ratio" := #"Maximum Flowrate Pump B" / #"Ratio/100";
END_REGION

REGION Network 4
   RUNG wire#powerrail
      { S7_Templates := "SrcType := Real" } LT_Contact(in1 := #"Mixing Ratio 100:B", in2 := #"Ratio margin")
      Move(in := #"Individual flowrate A MR", out1 => #"A Flowrate Compensated")
   END_RUNG
   RUNG wire#powerrail
      { S7_Templates := "SrcType := Real" } GE_Contact(in1 := #"Mixing Ratio 100:B", in2 := #"Ratio margin")
      Move(in := #"Flowrate A Per ratio", out1 => #"A Flowrate Compensated")
   END_RUNG
   // the same network as SCL:
   IF #"Mixing Ratio 100:B" < #"Ratio margin" THEN
       #"A Flowrate Compensated" := #"Individual flowrate A MR";
   END_IF;
   IF #"Mixing Ratio 100:B" >= #"Ratio margin" THEN
       #"A Flowrate Compensated" := #"Flowrate A Per ratio";
   END_IF;
END_REGION

REGION Network 5
   RUNG wire#powerrail
      Div(in1 := #"A Flowrate Compensated", in2 := 100.0, out => #"Individual flowrate B1 MR")
      Mul(in1 := #"Individual flowrate B1 MR", in2 := #"Mixing Ratio 100:B", out => #"Individual flowrate B MR")
   END_RUNG
   // the same network as SCL:
   #"Individual flowrate B1 MR" := #"A Flowrate Compensated" / 100.0;
   #"Individual flowrate B MR" := #"Individual flowrate B1 MR" * #"Mixing Ratio 100:B";
END_REGION

REGION Network 6: Mixed flowrate
   RUNG wire#powerrail
      Add(in1 := #"A Flowrate Compensated", in2 := #"Individual flowrate B MR", out => #"Mixed flowrate A+B")
      Move(in := #"Mixed flowrate A+B", out1 => #"Mixed Flowrate")
   END_RUNG
   // the same network as SCL:
   #"Mixed flowrate A+B" := #"A Flowrate Compensated" + #"Individual flowrate B MR";
   #"Mixed Flowrate" := #"Mixed flowrate A+B";
END_REGION

